LIN {X 0,Y 483.9,Z 922.544,A -85,B 0,C 180,E1 -6915.573,E2 -6915.573} C_VEL
LIN {X 0,Y 483.495,Z 935.94,A -85,B 0,C 180,E1 -6916.125,E2 -6916.125} C_VEL
LIN {X 0,Y 483.076,Z 947.548,A -85,B 0,C 180,E1 -6916.777,E2 -6916.777} C_VEL
LIN {X 0,Y 482.662,Z 958.984,A -85,B 0,C 180,E1 -6917.599,E2 -6917.599} C_VEL
LIN {X 0,Y 482.218,Z 969.588,A -85,B 0,C 180,E1 -6918.548,E2 -6918.548} C_VEL
LIN {X 0,Y 481.844,Z 978.283,A -85,B 0,C 180,E1 -6919.497,E2 -6919.497} C_VEL
LIN {X 0,Y 481.566,Z 986.33,A -85,B 0,C 180,E1 -6920.552,E2 -6920.552} C_VEL
LIN {X 0,Y 481.287,Z 994.208,A -85,B 0,C 180,E1 -6921.816,E2 -6921.816} C_VEL
LIN {X 0,Y 481.075,Z 1001.479,A -85,B 0,C 180,E1 -6923.29,E2 -6923.29} C_VEL
LIN {X 0,Y 481,Z 1006.335,A -85,B 0,C 180,E1 -6924.552,E2 -6924.552} C_VEL
LIN {X 0,Y 480.896,Z 1010.045,A -85,B 0,C 180,E1 -6925.811,E2 -6925.811} C_VEL
LIN {X 0,Y 480.923,Z 1011.97,A -85,B 0,C 180,E1 -6926.65,E2 -6926.65} C_VEL
LIN {X 0,Y 480.824,Z 1014.423,A -85,B 0,C 180,E1 -6928.326,E2 -6928.326} C_VEL
LIN {X 0,Y 480.773,Z 1015.041,A -85,B 0,C 180,E1 -6929.164,E2 -6929.164} C_VEL
LIN {X 0,Y 480.758,Z 1015.261,A -85,B 0,C 180,E1 -6930.001,E2 -6930.001} C_VEL
LIN {X 0,Y 480.773,Z 1015.039,A -85,B 0,C 180,E1 -6930.839,E2 -6930.839} C_VEL
LIN {X 0,Y 480.824,Z 1014.418,A -85,B 0,C 180,E1 -6931.677,E2 -6931.677} C_VEL
LIN {X 0,Y 480.924,Z 1011.961,A -85,B 0,C 180,E1 -6933.353,E2 -6933.353} C_VEL
LIN {X 0,Y 480.899,Z 1008.931,A -85,B 0,C 180,E1 -6934.612,E2 -6934.612} C_VEL
LIN {X 0,Y 481.047,Z 1004.858,A -85,B 0,C 180,E1 -6935.871,E2 -6935.871} C_VEL
LIN {X 0,Y 481.118,Z 998.567,A -85,B 0,C 180,E1 -6937.345,E2 -6937.345} C_VEL
LIN {X 0,Y 481.382,Z 991.735,A -85,B 0,C 180,E1 -6938.608,E2 -6938.608} C_VEL
LIN {X 0,Y 481.695,Z 983.271,A -85,B 0,C 180,E1 -6939.873,E2 -6939.873} C_VEL
LIN {X 0,Y 482.021,Z 974.606,A -85,B 0,C 180,E1 -6940.927,E2 -6940.927} C_VEL
LIN {X 0,Y 482.499,Z 963.942,A -85,B 0,C 180,E1 -6941.981,E2 -6941.981} C_VEL
LIN {X 0,Y 482.896,Z 952.218,A -85,B 0,C 180,E1 -6942.912,E2 -6942.912} C_VEL
LIN {X 0,Y 483.349,Z 939.937,A -85,B 0,C 180,E1 -6943.668,E2 -6943.668} C_VEL
LIN {X 0,Y 483.709,Z 927.469,A -85,B 0,C 180,E1 -6944.248,E2 -6944.248} C_VEL
LIN {X 0,Y 483.765,Z 919.717,A -85,B 0,C 180,E1 -6944.528,E2 -6944.528} C_VEL
LIN {X 0,Y 481.921,Z 906.606,A -85,B 0,C 180,E1 -6944.909,E2 -6944.909} C_VEL
LIN {X 0,Y 481.609,Z 903.06,A -85,B 0,C 180,E1 -6945.013,E2 -6945.013} C_VEL
LIN {X 0,Y 481.961,Z 889.747,A -85,B 0,C 180,E1 -6947.833,E2 -6947.833} C_VEL
LIN {X 0,Y 482.255,Z 874.313,A -85,B 0,C 180,E1 -6951.142,E2 -6951.142} C_VEL
LIN {X 0,Y 482.646,Z 860.861,A -85,B 0,C 180,E1 -6954.063,E2 -6954.063} C_VEL
LIN {X 0,Y 483.053,Z 846.87,A -85,B 0,C 180,E1 -6957.129,E2 -6957.129} C_VEL
LIN {X 0,Y 483.485,Z 831.351,A -85,B 0,C 180,E1 -6960.583,E2 -6960.583} C_VEL
LIN {X 0,Y 483.933,Z 818.655,A -85,B 0,C 180,E1 -6963.496,E2 -6963.496} C_VEL
LIN {X 0,Y 484.248,Z 807.022,A -85,B 0,C 180,E1 -6966.267,E2 -6966.267} C_VEL
LIN {X 0,Y 483.231,Z 800.666,A -85,B 0,C 180,E1 -6967.922,E2 -6967.922} C_VEL
LIN {X 0,Y 481.634,Z 792.492,A -85,B 0,C 180,E1 -6970.203,E2 -6970.203} C_VEL
LIN {X 0,Y 481.616,Z 792.493,A -85,B 0,C 180,E1 -6973.304,E2 -6973.304} C_VEL
LIN {X 0,Y 481.603,Z 792.499,A -85,B 0,C 180,E1 -6975.649,E2 -6975.649} C_VEL
LIN {X 0,Y 481.606,Z 792.492,A -85,B 0,C 180,E1 -6978.953,E2 -6978.953} C_VEL
LIN {X 0,Y 481.618,Z 792.494,A -85,B 0,C 180,E1 -6982,E2 -6982} C_VEL
LIN {X 0,Y 481.648,Z 792.488,A -85,B 0,C 180,E1 -6985.314,E2 -6985.314} C_VEL
LIN {X 0,Y 481.624,Z 792.492,A -85,B 0,C 180,E1 -6988.31,E2 -6988.31} C_VEL
LIN {X 0,Y 481.631,Z 792.488,A -85,B 0,C 180,E1 -6991.214,E2 -6991.214} C_VEL
LIN {X 0,Y 481.607,Z 792.496,A -85,B 0,C 180,E1 -6994.037,E2 -6994.037} C_VEL
LIN {X 0,Y 481.632,Z 792.488,A -85,B 0,C 180,E1 -6996.825,E2 -6996.825} C_VEL
LIN {X 0,Y 481.617,Z 792.491,A -85,B 0,C 180,E1 -6999.499,E2 -6999.499} C_VEL
LIN {X 0,Y 481.64,Z 792.493,A -85,B 0,C 180,E1 -7002.156,E2 -7002.156} C_VEL
LIN {X 0,Y 481.694,Z 792.486,A -85,B 0,C 180,E1 -7004.774,E2 -7004.774} C_VEL
LIN {X 0,Y 481.712,Z 792.618,A -85,B 0,C 180,E1 -7006.043,E2 -7006.043} C_VEL
LIN {X 0,Y 483.56,Z 799.412,A -85,B 0,C 180,E1 -7006.446,E2 -7006.446} C_VEL
LIN {X 0,Y 483.478,Z 810.921,A -85,B 0,C 180,E1 -7007.169,E2 -7007.169} C_VEL
LIN {X 0,Y 483.179,Z 820.671,A -85,B 0,C 180,E1 -7007.931,E2 -7007.931} C_VEL
LIN {X 0,Y 482.897,Z 828.589,A -85,B 0,C 180,E1 -7008.669,E2 -7008.669} C_VEL
LIN {X 0,Y 482.517,Z 837.913,A -85,B 0,C 180,E1 -7009.722,E2 -7009.722} C_VEL
LIN {X 0,Y 482.217,Z 845.434,A -85,B 0,C 180,E1 -7010.775,E2 -7010.775} C_VEL
LIN {X 0,Y 481.924,Z 851.738,A -85,B 0,C 180,E1 -7011.826,E2 -7011.826} C_VEL
LIN {X 0,Y 481.823,Z 856.164,A -85,B 0,C 180,E1 -7012.692,E2 -7012.692} C_VEL
LIN {X 0,Y 481.635,Z 862.067,A -85,B 0,C 180,E1 -7014.137,E2 -7014.137} C_VEL
LIN {X 0,Y 481.389,Z 864.819,A -85,B 0,C 180,E1 -7014.975,E2 -7014.975} C_VEL
LIN {X 0,Y 481.403,Z 866.963,A -85,B 0,C 180,E1 -7015.814,E2 -7015.814} C_VEL
LIN {X 0,Y 481.31,Z 870.195,A -85,B 0,C 180,E1 -7017.489,E2 -7017.489} C_VEL
LIN {X 0,Y 481.129,Z 871.712,A -85,B 0,C 180,E1 -7019.163,E2 -7019.163} C_VEL
LIN {X 0,Y 481.106,Z 871.896,A -85,B 0,C 180,E1 -7020,E2 -7020} C_VEL
LIN {X 0,Y 481.129,Z 871.66,A -85,B 0,C 180,E1 -7020.837,E2 -7020.837} C_VEL
LIN {X 0,Y 481.171,Z 869.996,A -85,B 0,C 180,E1 -7022.511,E2 -7022.511} C_VEL
LIN {X 0,Y 481.34,Z 866.697,A -85,B 0,C 180,E1 -7024.187,E2 -7024.187} C_VEL
LIN {X 0,Y 481.414,Z 863.086,A -85,B 0,C 180,E1 -7025.445,E2 -7025.445} C_VEL
LIN {X 0,Y 481.598,Z 858.349,A -85,B 0,C 180,E1 -7026.704,E2 -7026.704} C_VEL
LIN {X 0,Y 481.74,Z 853.505,A -85,B 0,C 180,E1 -7027.756,E2 -7027.756} C_VEL
LIN {X 0,Y 482.022,Z 846.333,A -85,B 0,C 180,E1 -7029.018,E2 -7029.018} C_VEL
LIN {X 0,Y 482.274,Z 838.919,A -85,B 0,C 180,E1 -7030.071,E2 -7030.071} C_VEL
LIN {X 0,Y 482.556,Z 831.974,A -85,B 0,C 180,E1 -7030.914,E2 -7030.914} C_VEL
LIN {X 0,Y 482.8,Z 823.76,A -85,B 0,C 180,E1 -7031.759,E2 -7031.759} C_VEL
LIN {X 0,Y 483.183,Z 813.877,A -85,B 0,C 180,E1 -7032.602,E2 -7032.602} C_VEL
LIN {X 0,Y 483.482,Z 803.895,A -85,B 0,C 180,E1 -7033.283,E2 -7033.283} C_VEL
LIN {X 0,Y 483.46,Z 799.397,A -85,B 0,C 180,E1 -7033.557,E2 -7033.557} C_VEL
LIN {X 0,Y 481.664,Z 792.488,A -85,B 0,C 180,E1 -7033.985,E2 -7033.985} C_VEL
LIN {X 0,Y 481.641,Z 792.489,A -85,B 0,C 180,E1 -7036.096,E2 -7036.096} C_VEL
LIN {X 0,Y 481.625,Z 792.487,A -85,B 0,C 180,E1 -7038.725,E2 -7038.725} C_VEL
LIN {X 0,Y 481.623,Z 792.489,A -85,B 0,C 180,E1 -7041.396,E2 -7041.396} C_VEL
LIN {X 0,Y 481.619,Z 792.49,A -85,B 0,C 180,E1 -7044.116,E2 -7044.116} C_VEL
LIN {X 0,Y 481.646,Z 792.482,A -85,B 0,C 180,E1 -7047.114,E2 -7047.114} C_VEL
LIN {X 0,Y 481.658,Z 792.489,A -85,B 0,C 180,E1 -7049.743,E2 -7049.743} C_VEL
LIN {X 0,Y 481.653,Z 792.479,A -85,B 0,C 180,E1 -7052.676,E2 -7052.676} C_VEL
LIN {X 0,Y 481.654,Z 792.483,A -85,B 0,C 180,E1 -7055.201,E2 -7055.201} C_VEL
LIN {X 0,Y 481.635,Z 792.49,A -85,B 0,C 180,E1 -7058.003,E2 -7058.003} C_VEL
LIN {X 0,Y 481.631,Z 792.485,A -85,B 0,C 180,E1 -7061.045,E2 -7061.045} C_VEL
LIN {X 0,Y 481.66,Z 792.485,A -85,B 0,C 180,E1 -7064.458,E2 -7064.458} C_VEL
LIN {X 0,Y 481.646,Z 792.489,A -85,B 0,C 180,E1 -7067.838,E2 -7067.838} C_VEL
LIN {X 0,Y 481.672,Z 792.481,A -85,B 0,C 180,E1 -7071.14,E2 -7071.14} C_VEL
LIN {X 0,Y 481.665,Z 792.483,A -85,B 0,C 180,E1 -7074.796,E2 -7074.796} C_VEL
LIN {X 0,Y 481.662,Z 792.485,A -85,B 0,C 180,E1 -7077.81,E2 -7077.81} C_VEL
LIN {X 0,Y 481.704,Z 792.474,A -85,B 0,C 180,E1 -7081.218,E2 -7081.218} C_VEL
LIN {X 0,Y 481.675,Z 792.482,A -85,B 0,C 180,E1 -7084.115,E2 -7084.115} C_VEL
LIN {X 0,Y 480.993,Z 792.565,A -85,B 0,C 180,E1 -7084.813,E2 -7084.813} C_VEL
LIN {X 0,Y 478.124,Z 792.922,A -85,B 0,C 180,E1 -7085.947,E2 -7085.947} C_VEL
LIN {X 0,Y 475.706,Z 793.227,A -85,B 0,C 180,E1 -7086.861,E2 -7086.861} C_VEL
LIN {X 0,Y 474.67,Z 793.354,A -85,B 0,C 180,E1 -7087.568,E2 -7087.568} C_VEL
LIN {X 0,Y 474.586,Z 793.366,A -85,B 0,C 180,E1 -7087.807,E2 -7087.807} C_VEL
LIN {X 0,Y 474.66,Z 793.361,A -85,B 0,C 180,E1 -7090.088,E2 -7090.088} C_VEL
LIN {X 0,Y 474.642,Z 793.365,A -85,B 0,C 180,E1 -7092.773,E2 -7092.773} C_VEL
LIN {X 0,Y 474.674,Z 793.357,A -85,B 0,C 180,E1 -7095.612,E2 -7095.612} C_VEL
LIN {X 0,Y 477.158,Z 802.152,A -85,B 0,C 180,E1 -7096.151,E2 -7096.151} C_VEL
LIN {X 0,Y 477.085,Z 812.643,A -85,B 0,C 180,E1 -7096.812,E2 -7096.812} C_VEL
LIN {X 0,Y 476.651,Z 823.432,A -85,B 0,C 180,E1 -7097.654,E2 -7097.654} C_VEL
LIN {X 0,Y 476.309,Z 832.277,A -85,B 0,C 180,E1 -7098.509,E2 -7098.509} C_VEL
LIN {X 0,Y 475.895,Z 841.339,A -85,B 0,C 180,E1 -7099.576,E2 -7099.576} C_VEL
LIN {X 0,Y 475.468,Z 850.111,A -85,B 0,C 180,E1 -7100.856,E2 -7100.856} C_VEL
LIN {X 0,Y 475.125,Z 857.159,A -85,B 0,C 180,E1 -7102.134,E2 -7102.134} C_VEL
LIN {X 0,Y 475.013,Z 861.893,A -85,B 0,C 180,E1 -7103.201,E2 -7103.201} C_VEL
LIN {X 0,Y 474.635,Z 866.527,A -85,B 0,C 180,E1 -7104.475,E2 -7104.475} C_VEL
LIN {X 0,Y 474.515,Z 870.043,A -85,B 0,C 180,E1 -7105.752,E2 -7105.752} C_VEL
LIN {X 0,Y 474.413,Z 871.866,A -85,B 0,C 180,E1 -7106.601,E2 -7106.601} C_VEL
LIN {X 0,Y 474.428,Z 873.229,A -85,B 0,C 180,E1 -7107.451,E2 -7107.451} C_VEL
LIN {X 0,Y 474.342,Z 874.81,A -85,B 0,C 180,E1 -7109.15,E2 -7109.15} C_VEL
LIN {X 0,Y 474.361,Z 875.038,A -85,B 0,C 180,E1 -7109.998,E2 -7109.998} C_VEL
LIN {X 0,Y 474.305,Z 874.304,A -85,B 0,C 180,E1 -7111.697,E2 -7111.697} C_VEL
LIN {X 0,Y 474.427,Z 873.352,A -85,B 0,C 180,E1 -7112.546,E2 -7112.546} C_VEL
LIN {X 0,Y 474.408,Z 872.043,A -85,B 0,C 180,E1 -7113.396,E2 -7113.396} C_VEL
LIN {X 0,Y 474.554,Z 869.241,A -85,B 0,C 180,E1 -7114.671,E2 -7114.671} C_VEL
LIN {X 0,Y 474.825,Z 865.428,A -85,B 0,C 180,E1 -7115.945,E2 -7115.945} C_VEL
LIN {X 0,Y 475.021,Z 860.484,A -85,B 0,C 180,E1 -7117.234,E2 -7117.234} C_VEL
LIN {X 0,Y 475.259,Z 854.356,A -85,B 0,C 180,E1 -7118.502,E2 -7118.502} C_VEL
LIN {X 0,Y 475.672,Z 846.595,A -85,B 0,C 180,E1 -7119.781,E2 -7119.781} C_VEL
LIN {X 0,Y 476.051,Z 838.675,A -85,B 0,C 180,E1 -7120.848,E2 -7120.848} C_VEL
LIN {X 0,Y 476.451,Z 828.997,A -85,B 0,C 180,E1 -7121.916,E2 -7121.916} C_VEL
LIN {X 0,Y 476.812,Z 819.458,A -85,B 0,C 180,E1 -7122.772,E2 -7122.772} C_VEL
LIN {X 0,Y 477.177,Z 808.266,A -85,B 0,C 180,E1 -7123.573,E2 -7123.573} C_VEL
LIN {X 0,Y 477.358,Z 803.815,A -85,B 0,C 180,E1 -7123.84,E2 -7123.84} C_VEL
LIN {X 0,Y 475.979,Z 797.969,A -85,B 0,C 180,E1 -7124.208,E2 -7124.208} C_VEL
LIN {X 0,Y 474.653,Z 793.36,A -85,B 0,C 180,E1 -7124.495,E2 -7124.495} C_VEL
LIN {X 0,Y 474.65,Z 793.361,A -85,B 0,C 180,E1 -7127.224,E2 -7127.224} C_VEL
LIN {X 0,Y 474.655,Z 793.362,A -85,B 0,C 180,E1 -7129.908,E2 -7129.908} C_VEL
LIN {X 0,Y 474.633,Z 793.361,A -85,B 0,C 180,E1 -7133.357,E2 -7133.357} C_VEL
LIN {X 0,Y 474.657,Z 793.358,A -85,B 0,C 180,E1 -7136.37,E2 -7136.37} C_VEL
LIN {X 0,Y 474.618,Z 793.361,A -85,B 0,C 180,E1 -7139.25,E2 -7139.25} C_VEL
LIN {X 0,Y 474.611,Z 793.365,A -85,B 0,C 180,E1 -7142.429,E2 -7142.429} C_VEL
LIN {X 0,Y 474.612,Z 793.362,A -85,B 0,C 180,E1 -7145.468,E2 -7145.468} C_VEL
LIN {X 0,Y 474.615,Z 793.366,A -85,B 0,C 180,E1 -7148.454,E2 -7148.454} C_VEL
LIN {X 0,Y 474.637,Z 793.358,A -85,B 0,C 180,E1 -7150.96,E2 -7150.96} C_VEL
LIN {X 0,Y 474.608,Z 793.367,A -85,B 0,C 180,E1 -7154.102,E2 -7154.102} C_VEL
LIN {X 0,Y 474.641,Z 793.355,A -85,B 0,C 180,E1 -7157.068,E2 -7157.068} C_VEL
LIN {X 0,Y 474.662,Z 793.361,A -85,B 0,C 180,E1 -7160.456,E2 -7160.456} C_VEL
LIN {X 0,Y 474.58,Z 793.364,A -85,B 0,C 180,E1 -7163.675,E2 -7163.675} C_VEL
LIN {X 0,Y 474.629,Z 793.365,A -85,B 0,C 180,E1 -7166.779,E2 -7166.779} C_VEL
LIN {X 0,Y 474.599,Z 793.359,A -85,B 0,C 180,E1 -7169.769,E2 -7169.769} C_VEL
LIN {X 0,Y 474.699,Z 793.357,A -85,B 0,C 180,E1 -7172.68,E2 -7172.68} C_VEL
LIN {X 0,Y 474.644,Z 793.357,A -85,B 0,C 180,E1 -7175.506,E2 -7175.506} C_VEL
LIN {X 0,Y 474.654,Z 793.359,A -85,B 0,C 180,E1 -7179.184,E2 -7179.184} C_VEL
LIN {X 0,Y 474.64,Z 793.357,A -85,B 0,C 180,E1 -7181.884,E2 -7181.884} C_VEL
LIN {X 0,Y 474.682,Z 793.35,A -85,B 0,C 180,E1 -7184.544,E2 -7184.544} C_VEL
LIN {X 0,Y 474.724,Z 793.347,A -85,B 0,C 180,E1 -7188.038,E2 -7188.038} C_VEL
LIN {X 0,Y 474.712,Z 793.354,A -85,B 0,C 180,E1 -7191.486,E2 -7191.486} C_VEL
LIN {X 0,Y 474.753,Z 793.345,A -85,B 0,C 180,E1 -7194.052,E2 -7194.052} C_VEL
LIN {X 0,Y 474.876,Z 793.334,A -85,B 0,C 180,E1 -7197.455,E2 -7197.455} C_VEL
LIN {X 0,Y 474.89,Z 793.33,A -85,B 0,C 180,E1 -7200,E2 -7200} C_VEL
LIN {X 0,Y 474.875,Z 793.329,A -85,B 0,C 180,E1 -7202.545,E2 -7202.545} C_VEL
LIN {X 0,Y 474.74,Z 793.349,A -85,B 0,C 180,E1 -7205.948,E2 -7205.948} C_VEL
LIN {X 0,Y 474.709,Z 793.348,A -85,B 0,C 180,E1 -7208.514,E2 -7208.514} C_VEL
LIN {X 0,Y 474.721,Z 793.35,A -85,B 0,C 180,E1 -7211.962,E2 -7211.962} C_VEL
LIN {X 0,Y 474.661,Z 793.362,A -85,B 0,C 180,E1 -7215.768,E2 -7215.768} C_VEL
LIN {X 0,Y 474.645,Z 793.357,A -85,B 0,C 180,E1 -7219.011,E2 -7219.011} C_VEL
LIN {X 0,Y 474.571,Z 793.371,A -85,B 0,C 180,E1 -7221.73,E2 -7221.73} C_VEL
LIN {X 0,Y 474.614,Z 793.363,A -85,B 0,C 180,E1 -7224.495,E2 -7224.495} C_VEL
LIN {X 0,Y 474.62,Z 793.359,A -85,B 0,C 180,E1 -7227.325,E2 -7227.325} C_VEL
LIN {X 0,Y 474.587,Z 793.37,A -85,B 0,C 180,E1 -7230.232,E2 -7230.232} C_VEL
LIN {X 0,Y 474.606,Z 793.362,A -85,B 0,C 180,E1 -7233.223,E2 -7233.223} C_VEL
LIN {X 0,Y 474.564,Z 793.375,A -85,B 0,C 180,E1 -7236.326,E2 -7236.326} C_VEL
LIN {X 0,Y 474.587,Z 793.366,A -85,B 0,C 180,E1 -7239.645,E2 -7239.645} C_VEL
LIN {X 0,Y 474.561,Z 793.373,A -85,B 0,C 180,E1 -7242.94,E2 -7242.94} C_VEL
LIN {X 0,Y 474.585,Z 793.368,A -85,B 0,C 180,E1 -7245.895,E2 -7245.895} C_VEL
LIN {X 0,Y 474.602,Z 793.368,A -85,B 0,C 180,E1 -7249.47,E2 -7249.47} C_VEL
LIN {X 0,Y 474.618,Z 793.527,A -85,B 0,C 180,E1 -7249.597,E2 -7249.597} C_VEL
LIN {X 0,Y 476.953,Z 805.247,A -85,B 0,C 180,E1 -7252.835,E2 -7252.835} C_VEL
LIN {X 0,Y 477.313,Z 810.127,A -85,B 0,C 180,E1 -7254.079,E2 -7254.079} C_VEL
LIN {X 0,Y 476.863,Z 822.093,A -85,B 0,C 180,E1 -7256.957,E2 -7256.957} C_VEL
LIN {X 0,Y 476.399,Z 834.791,A -85,B 0,C 180,E1 -7259.898,E2 -7259.898} C_VEL
LIN {X 0,Y 476.003,Z 848.539,A -85,B 0,C 180,E1 -7263.001,E2 -7263.001} C_VEL
LIN {X 0,Y 475.588,Z 862.135,A -85,B 0,C 180,E1 -7266.023,E2 -7266.023} C_VEL
LIN {X 0,Y 475.137,Z 877.652,A -85,B 0,C 180,E1 -7269.435,E2 -7269.435} C_VEL
LIN {X 0,Y 474.809,Z 891.946,A -85,B 0,C 180,E1 -7272.56,E2 -7272.56} C_VEL
LIN {X 0,Y 474.543,Z 902.182,A -85,B 0,C 180,E1 -7274.788,E2 -7274.788} C_VEL
LIN {X 0,Y 475.988,Z 914.958,A -85,B 0,C 180,E1 -7275.123,E2 -7275.123} C_VEL
LIN {X 0,Y 476.932,Z 923.027,A -85,B 0,C 180,E1 -7275.412,E2 -7275.412} C_VEL
LIN {X 0,Y 476.524,Z 935.928,A -85,B 0,C 180,E1 -7275.972,E2 -7275.972} C_VEL
LIN {X 0,Y 476.038,Z 948.259,A -85,B 0,C 180,E1 -7276.697,E2 -7276.697} C_VEL
LIN {X 0,Y 475.624,Z 959.269,A -85,B 0,C 180,E1 -7277.523,E2 -7277.523} C_VEL
LIN {X 0,Y 475.139,Z 969.601,A -85,B 0,C 180,E1 -7278.483,E2 -7278.483} C_VEL
LIN {X 0,Y 474.734,Z 978.948,A -85,B 0,C 180,E1 -7279.553,E2 -7279.553} C_VEL
LIN {X 0,Y 474.405,Z 988.081,A -85,B 0,C 180,E1 -7280.838,E2 -7280.838} C_VEL
LIN {X 0,Y 474.143,Z 995.45,A -85,B 0,C 180,E1 -7282.121,E2 -7282.121} C_VEL
LIN {X 0,Y 473.979,Z 1001.499,A -85,B 0,C 180,E1 -7283.442,E2 -7283.442} C_VEL
LIN {X 0,Y 473.893,Z 1006.643,A -85,B 0,C 180,E1 -7284.897,E2 -7284.897} C_VEL
LIN {X 0,Y 473.85,Z 1009.008,A -85,B 0,C 180,E1 -7285.749,E2 -7285.749} C_VEL
LIN {X 0,Y 473.881,Z 1010.935,A -85,B 0,C 180,E1 -7286.601,E2 -7286.601} C_VEL
LIN {X 0,Y 473.792,Z 1013.39,A -85,B 0,C 180,E1 -7288.302,E2 -7288.302} C_VEL
LIN {X 0,Y 473.747,Z 1014.009,A -85,B 0,C 180,E1 -7289.152,E2 -7289.152} C_VEL
LIN {X 0,Y 473.734,Z 1014.229,A -85,B 0,C 180,E1 -7290.002,E2 -7290.002} C_VEL
LIN {X 0,Y 473.747,Z 1014.007,A -85,B 0,C 180,E1 -7290.852,E2 -7290.852} C_VEL
LIN {X 0,Y 473.793,Z 1013.385,A -85,B 0,C 180,E1 -7291.702,E2 -7291.702} C_VEL
LIN {X 0,Y 473.882,Z 1010.925,A -85,B 0,C 180,E1 -7293.402,E2 -7293.402} C_VEL
LIN {X 0,Y 473.86,Z 1007.894,A -85,B 0,C 180,E1 -7294.68,E2 -7294.68} C_VEL
LIN {X 0,Y 473.989,Z 1003.816,A -85,B 0,C 180,E1 -7295.959,E2 -7295.959} C_VEL
LIN {X 0,Y 474.079,Z 997.525,A -85,B 0,C 180,E1 -7297.455,E2 -7297.455} C_VEL
LIN {X 0,Y 474.333,Z 990.688,A -85,B 0,C 180,E1 -7298.737,E2 -7298.737} C_VEL
LIN {X 0,Y 474.628,Z 982.217,A -85,B 0,C 180,E1 -7300.021,E2 -7300.021} C_VEL
LIN {X 0,Y 475.01,Z 973.557,A -85,B 0,C 180,E1 -7301.091,E2 -7301.091} C_VEL
LIN {X 0,Y 475.52,Z 962.895,A -85,B 0,C 180,E1 -7302.159,E2 -7302.159} C_VEL
LIN {X 0,Y 475.901,Z 951.335,A -85,B 0,C 180,E1 -7303.092,E2 -7303.092} C_VEL
LIN {X 0,Y 476.385,Z 938.884,A -85,B 0,C 180,E1 -7303.872,E2 -7303.872} C_VEL
LIN {X 0,Y 476.79,Z 926.421,A -85,B 0,C 180,E1 -7304.459,E2 -7304.459} C_VEL
LIN {X 0,Y 476.773,Z 920.23,A -85,B 0,C 180,E1 -7304.691,E2 -7304.691} C_VEL
LIN {X 0,Y 475.08,Z 907.695,A -85,B 0,C 180,E1 -7305.087,E2 -7305.087} C_VEL
LIN {X 0,Y 474.548,Z 902.188,A -85,B 0,C 180,E1 -7305.215,E2 -7305.215} C_VEL
LIN {X 0,Y 474.929,Z 887.43,A -85,B 0,C 180,E1 -7308.416,E2 -7308.416} C_VEL
LIN {X 0,Y 475.218,Z 874.257,A -85,B 0,C 180,E1 -7311.297,E2 -7311.297} C_VEL
LIN {X 0,Y 475.622,Z 861.091,A -85,B 0,C 180,E1 -7314.209,E2 -7314.209} C_VEL
LIN {X 0,Y 476.027,Z 847.465,A -85,B 0,C 180,E1 -7317.239,E2 -7317.239} C_VEL
LIN {X 0,Y 476.482,Z 832.656,A -85,B 0,C 180,E1 -7320.59,E2 -7320.59} C_VEL
LIN {X 0,Y 476.977,Z 819.963,A -85,B 0,C 180,E1 -7323.543,E2 -7323.543} C_VEL
LIN {X 0,Y 477.336,Z 808.396,A -85,B 0,C 180,E1 -7326.344,E2 -7326.344} C_VEL
LIN {X 0,Y 476.279,Z 802.037,A -85,B 0,C 180,E1 -7328.03,E2 -7328.03} C_VEL
LIN {X 0,Y 474.597,Z 793.369,A -85,B 0,C 180,E1 -7330.471,E2 -7330.471} C_VEL
LIN {X 0,Y 474.562,Z 793.371,A -85,B 0,C 180,E1 -7333.476,E2 -7333.476} C_VEL
LIN {X 0,Y 474.546,Z 793.371,A -85,B 0,C 180,E1 -7336.527,E2 -7336.527} C_VEL
LIN {X 0,Y 474.571,Z 793.373,A -85,B 0,C 180,E1 -7339.337,E2 -7339.337} C_VEL
LIN {X 0,Y 474.583,Z 793.37,A -85,B 0,C 180,E1 -7341.71,E2 -7341.71} C_VEL
LIN {X 0,Y 474.571,Z 793.367,A -85,B 0,C 180,E1 -7344.721,E2 -7344.721} C_VEL
LIN {X 0,Y 474.614,Z 793.366,A -85,B 0,C 180,E1 -7347.786,E2 -7347.786} C_VEL
LIN {X 0,Y 474.577,Z 793.367,A -85,B 0,C 180,E1 -7350.897,E2 -7350.897} C_VEL
LIN {X 0,Y 474.559,Z 793.372,A -85,B 0,C 180,E1 -7353.622,E2 -7353.622} C_VEL
LIN {X 0,Y 474.599,Z 793.366,A -85,B 0,C 180,E1 -7356.654,E2 -7356.654} C_VEL
LIN {X 0,Y 474.618,Z 793.363,A -85,B 0,C 180,E1 -7359.183,E2 -7359.183} C_VEL
LIN {X 0,Y 474.594,Z 793.369,A -85,B 0,C 180,E1 -7361.882,E2 -7361.882} C_VEL
LIN {X 0,Y 474.654,Z 793.364,A -85,B 0,C 180,E1 -7364.543,E2 -7364.543} C_VEL
LIN {X 0,Y 474.638,Z 793.364,A -85,B 0,C 180,E1 -7365.804,E2 -7365.804} C_VEL
LIN {X 0,Y 476.853,Z 802.263,A -85,B 0,C 180,E1 -7366.36,E2 -7366.36} C_VEL
LIN {X 0,Y 476.602,Z 813.02,A -85,B 0,C 180,E1 -7367.063,E2 -7367.063} C_VEL
LIN {X 0,Y 476.258,Z 822.874,A -85,B 0,C 180,E1 -7367.861,E2 -7367.861} C_VEL
LIN {X 0,Y 476.029,Z 829.646,A -85,B 0,C 180,E1 -7368.503,E2 -7368.503} C_VEL
LIN {X 0,Y 475.628,Z 838.964,A -85,B 0,C 180,E1 -7369.571,E2 -7369.571} C_VEL
LIN {X 0,Y 475.289,Z 846.504,A -85,B 0,C 180,E1 -7370.639,E2 -7370.639} C_VEL
LIN {X 0,Y 474.979,Z 852.816,A -85,B 0,C 180,E1 -7371.705,E2 -7371.705} C_VEL
LIN {X 0,Y 474.865,Z 857.199,A -85,B 0,C 180,E1 -7372.573,E2 -7372.573} C_VEL
LIN {X 0,Y 474.662,Z 863.15,A -85,B 0,C 180,E1 -7374.051,E2 -7374.051} C_VEL
LIN {X 0,Y 474.402,Z 865.908,A -85,B 0,C 180,E1 -7374.9,E2 -7374.9} C_VEL
LIN {X 0,Y 474.404,Z 868.049,A -85,B 0,C 180,E1 -7375.752,E2 -7375.752} C_VEL
LIN {X 0,Y 474.31,Z 871.277,A -85,B 0,C 180,E1 -7377.452,E2 -7377.452} C_VEL
LIN {X 0,Y 474.115,Z 872.783,A -85,B 0,C 180,E1 -7379.151,E2 -7379.151} C_VEL
LIN {X 0,Y 474.09,Z 872.959,A -85,B 0,C 180,E1 -7380,E2 -7380} C_VEL
LIN {X 0,Y 474.115,Z 872.714,A -85,B 0,C 180,E1 -7380.849,E2 -7380.849} C_VEL
LIN {X 0,Y 474.154,Z 871.025,A -85,B 0,C 180,E1 -7382.549,E2 -7382.549} C_VEL
LIN {X 0,Y 474.33,Z 867.692,A -85,B 0,C 180,E1 -7384.249,E2 -7384.249} C_VEL
LIN {X 0,Y 474.421,Z 864.051,A -85,B 0,C 180,E1 -7385.526,E2 -7385.526} C_VEL
LIN {X 0,Y 474.617,Z 859.281,A -85,B 0,C 180,E1 -7386.803,E2 -7386.803} C_VEL
LIN {X 0,Y 474.776,Z 854.405,A -85,B 0,C 180,E1 -7387.87,E2 -7387.87} C_VEL
LIN {X 0,Y 475.077,Z 847.198,A -85,B 0,C 180,E1 -7389.151,E2 -7389.151} C_VEL
LIN {X 0,Y 475.34,Z 839.741,A -85,B 0,C 180,E1 -7390.22,E2 -7390.22} C_VEL
LIN {X 0,Y 475.641,Z 832.756,A -85,B 0,C 180,E1 -7391.075,E2 -7391.075} C_VEL
LIN {X 0,Y 475.896,Z 824.497,A -85,B 0,C 180,E1 -7391.932,E2 -7391.932} C_VEL
LIN {X 0,Y 476.351,Z 813.356,A -85,B 0,C 180,E1 -7392.883,E2 -7392.883} C_VEL
LIN {X 0,Y 476.655,Z 803.186,A -85,B 0,C 180,E1 -7393.559,E2 -7393.559} C_VEL
LIN {X 0,Y 476.406,Z 800.049,A -85,B 0,C 180,E1 -7393.761,E2 -7393.761} C_VEL
LIN {X 0,Y 474.639,Z 793.362,A -85,B 0,C 180,E1 -7394.196,E2 -7394.196} C_VEL
LIN {X 0,Y 474.592,Z 793.365,A -85,B 0,C 180,E1 -7396.342,E2 -7396.342} C_VEL
LIN {X 0,Y 474.582,Z 793.365,A -85,B 0,C 180,E1 -7399.014,E2 -7399.014} C_VEL
LIN {X 0,Y 474.572,Z 793.369,A -85,B 0,C 180,E1 -7401.73,E2 -7401.73} C_VEL
LIN {X 0,Y 474.586,Z 793.364,A -85,B 0,C 180,E1 -7404.497,E2 -7404.497} C_VEL
LIN {X 0,Y 474.598,Z 793.361,A -85,B 0,C 180,E1 -7407.327,E2 -7407.327} C_VEL
LIN {X 0,Y 474.589,Z 793.365,A -85,B 0,C 180,E1 -7410.231,E2 -7410.231} C_VEL
LIN {X 0,Y 474.618,Z 793.356,A -85,B 0,C 180,E1 -7413.222,E2 -7413.222} C_VEL
LIN {X 0,Y 474.575,Z 793.366,A -85,B 0,C 180,E1 -7416.325,E2 -7416.325} C_VEL
LIN {X 0,Y 474.606,Z 793.364,A -85,B 0,C 180,E1 -7419.643,E2 -7419.643} C_VEL
LIN {X 0,Y 474.58,Z 793.363,A -85,B 0,C 180,E1 -7422.938,E2 -7422.938} C_VEL
LIN {X 0,Y 474.609,Z 793.367,A -85,B 0,C 180,E1 -7425.894,E2 -7425.894} C_VEL
LIN {X 0,Y 474.613,Z 793.36,A -85,B 0,C 180,E1 -7429.043,E2 -7429.043} C_VEL
LIN {X 0,Y 474.612,Z 793.364,A -85,B 0,C 180,E1 -7431.704,E2 -7431.704} C_VEL
LIN {X 0,Y 474.627,Z 793.361,A -85,B 0,C 180,E1 -7434.725,E2 -7434.725} C_VEL
LIN {X 0,Y 474.641,Z 793.359,A -85,B 0,C 180,E1 -7437.787,E2 -7437.787} C_VEL
LIN {X 0,Y 474.628,Z 793.357,A -85,B 0,C 180,E1 -7440.884,E2 -7440.884} C_VEL
LIN {X 0,Y 474.633,Z 793.356,A -85,B 0,C 180,E1 -7443.626,E2 -7443.626} C_VEL
LIN {X 0,Y 474.64,Z 793.363,A -85,B 0,C 180,E1 -7446.641,E2 -7446.641} C_VEL
LIN {X 0,Y 474.586,Z 793.366,A -85,B 0,C 180,E1 -7447.807,E2 -7447.807} C_VEL
LIN {X 0,Y 473.921,Z 793.455,A -85,B 0,C 180,E1 -7448.515,E2 -7448.515} C_VEL
LIN {X 0,Y 471.082,Z 793.807,A -85,B 0,C 180,E1 -7449.666,E2 -7449.666} C_VEL
LIN {X 0,Y 468.698,Z 794.107,A -85,B 0,C 180,E1 -7450.594,E2 -7450.594} C_VEL
LIN {X 0,Y 467.697,Z 794.227,A -85,B 0,C 180,E1 -7451.311,E2 -7451.311} C_VEL
LIN {X 0,Y 467.627,Z 794.235,A -85,B 0,C 180,E1 -7451.553,E2 -7451.553} C_VEL
LIN {X 0,Y 467.645,Z 794.235,A -85,B 0,C 180,E1 -7454.304,E2 -7454.304} C_VEL
LIN {X 0,Y 467.649,Z 794.397,A -85,B 0,C 180,E1 -7455.391,E2 -7455.391} C_VEL
LIN {X 0,Y 470.186,Z 803.216,A -85,B 0,C 180,E1 -7455.941,E2 -7455.941} C_VEL
LIN {X 0,Y 470.431,Z 806.901,A -85,B 0,C 180,E1 -7456.169,E2 -7456.169} C_VEL
LIN {X 0,Y 470.131,Z 817.479,A -85,B 0,C 180,E1 -7456.898,E2 -7456.898} C_VEL
LIN {X 0,Y 469.646,Z 827.956,A -85,B 0,C 180,E1 -7457.796,E2 -7457.796} C_VEL
LIN {X 0,Y 469.244,Z 837.16,A -85,B 0,C 180,E1 -7458.771,E2 -7458.771} C_VEL
LIN {X 0,Y 468.836,Z 845.541,A -85,B 0,C 180,E1 -7459.854,E2 -7459.854} C_VEL
LIN {X 0,Y 468.367,Z 853.668,A -85,B 0,C 180,E1 -7461.151,E2 -7461.151} C_VEL
LIN {X 0,Y 468.089,Z 859.443,A -85,B 0,C 180,E1 -7462.284,E2 -7462.284} C_VEL
LIN {X 0,Y 467.961,Z 864.59,A -85,B 0,C 180,E1 -7463.531,E2 -7463.531} C_VEL
LIN {X 0,Y 467.559,Z 868.851,A -85,B 0,C 180,E1 -7464.824,E2 -7464.824} C_VEL
LIN {X 0,Y 467.509,Z 871.075,A -85,B 0,C 180,E1 -7465.688,E2 -7465.688} C_VEL
LIN {X 0,Y 467.402,Z 872.898,A -85,B 0,C 180,E1 -7466.55,E2 -7466.55} C_VEL
LIN {X 0,Y 467.418,Z 874.26,A -85,B 0,C 180,E1 -7467.413,E2 -7467.413} C_VEL
LIN {X 0,Y 467.333,Z 875.839,A -85,B 0,C 180,E1 -7469.137,E2 -7469.137} C_VEL
LIN {X 0,Y 467.347,Z 876.068,A -85,B 0,C 180,E1 -7469.998,E2 -7469.998} C_VEL
LIN {X 0,Y 467.289,Z 875.334,A -85,B 0,C 180,E1 -7471.722,E2 -7471.722} C_VEL
LIN {X 0,Y 467.416,Z 874.381,A -85,B 0,C 180,E1 -7472.584,E2 -7472.584} C_VEL
LIN {X 0,Y 467.396,Z 873.073,A -85,B 0,C 180,E1 -7473.447,E2 -7473.447} C_VEL
LIN {X 0,Y 467.551,Z 870.272,A -85,B 0,C 180,E1 -7474.741,E2 -7474.741} C_VEL
LIN {X 0,Y 467.85,Z 866.456,A -85,B 0,C 180,E1 -7476.034,E2 -7476.034} C_VEL
LIN {X 0,Y 468.063,Z 861.459,A -85,B 0,C 180,E1 -7477.355,E2 -7477.355} C_VEL
LIN {X 0,Y 468.319,Z 855.384,A -85,B 0,C 180,E1 -7478.629,E2 -7478.629} C_VEL
LIN {X 0,Y 468.754,Z 847.622,A -85,B 0,C 180,E1 -7479.927,E2 -7479.927} C_VEL
LIN {X 0,Y 469.158,Z 839.702,A -85,B 0,C 180,E1 -7481.009,E2 -7481.009} C_VEL
LIN {X 0,Y 469.58,Z 830.024,A -85,B 0,C 180,E1 -7482.093,E2 -7482.093} C_VEL
LIN {X 0,Y 469.966,Z 820.484,A -85,B 0,C 180,E1 -7482.961,E2 -7482.961} C_VEL
LIN {X 0,Y 470.35,Z 809.276,A -85,B 0,C 180,E1 -7483.775,E2 -7483.775} C_VEL
LIN {X 0,Y 470.511,Z 804.842,A -85,B 0,C 180,E1 -7484.046,E2 -7484.046} C_VEL
LIN {X 0,Y 467.626,Z 794.235,A -85,B 0,C 180,E1 -7484.718,E2 -7484.718} C_VEL
LIN {X 0,Y 467.608,Z 794.241,A -85,B 0,C 180,E1 -7487.491,E2 -7487.491} C_VEL
LIN {X 0,Y 467.622,Z 794.234,A -85,B 0,C 180,E1 -7490.221,E2 -7490.221} C_VEL
LIN {X 0,Y 467.571,Z 794.245,A -85,B 0,C 180,E1 -7493.941,E2 -7493.941} C_VEL
LIN {X 0,Y 467.612,Z 794.233,A -85,B 0,C 180,E1 -7496.798,E2 -7496.798} C_VEL
LIN {X 0,Y 467.551,Z 794.246,A -85,B 0,C 180,E1 -7499.736,E2 -7499.736} C_VEL
LIN {X 0,Y 467.578,Z 794.238,A -85,B 0,C 180,E1 -7502.756,E2 -7502.756} C_VEL
LIN {X 0,Y 467.549,Z 794.247,A -85,B 0,C 180,E1 -7505.888,E2 -7505.888} C_VEL
LIN {X 0,Y 467.591,Z 794.236,A -85,B 0,C 180,E1 -7509.141,E2 -7509.141} C_VEL
LIN {X 0,Y 467.609,Z 794.238,A -85,B 0,C 180,E1 -7512.57,E2 -7512.57} C_VEL
LIN {X 0,Y 467.564,Z 794.245,A -85,B 0,C 180,E1 -7516.175,E2 -7516.175} C_VEL
LIN {X 0,Y 467.578,Z 794.242,A -85,B 0,C 180,E1 -7518.72,E2 -7518.72} C_VEL
LIN {X 0,Y 467.566,Z 794.236,A -85,B 0,C 180,E1 -7521.405,E2 -7521.405} C_VEL
LIN {X 0,Y 467.55,Z 794.244,A -85,B 0,C 180,E1 -7524.259,E2 -7524.259} C_VEL
LIN {X 0,Y 467.568,Z 794.239,A -85,B 0,C 180,E1 -7527.319,E2 -7527.319} C_VEL
LIN {X 0,Y 467.563,Z 794.243,A -85,B 0,C 180,E1 -7530.664,E2 -7530.664} C_VEL
LIN {X 0,Y 467.612,Z 794.234,A -85,B 0,C 180,E1 -7533.199,E2 -7533.199} C_VEL
LIN {X 0,Y 467.577,Z 794.239,A -85,B 0,C 180,E1 -7536.467,E2 -7536.467} C_VEL
LIN {X 0,Y 467.606,Z 794.232,A -85,B 0,C 180,E1 -7539.776,E2 -7539.776} C_VEL
LIN {X 0,Y 467.592,Z 794.237,A -85,B 0,C 180,E1 -7542.506,E2 -7542.506} C_VEL
LIN {X 0,Y 467.589,Z 794.239,A -85,B 0,C 180,E1 -7545.196,E2 -7545.196} C_VEL
LIN {X 0,Y 467.667,Z 794.227,A -85,B 0,C 180,E1 -7547.855,E2 -7547.855} C_VEL
LIN {X 0,Y 467.666,Z 794.231,A -85,B 0,C 180,E1 -7551.357,E2 -7551.357} C_VEL
LIN {X 0,Y 467.718,Z 794.222,A -85,B 0,C 180,E1 -7553.962,E2 -7553.962} C_VEL
LIN {X 0,Y 467.841,Z 794.21,A -85,B 0,C 180,E1 -7557.417,E2 -7557.417} C_VEL
LIN {X 0,Y 467.862,Z 794.205,A -85,B 0,C 180,E1 -7560,E2 -7560} C_VEL
LIN {X 0,Y 467.841,Z 794.206,A -85,B 0,C 180,E1 -7562.583,E2 -7562.583} C_VEL
LIN {X 0,Y 467.702,Z 794.224,A -85,B 0,C 180,E1 -7566.038,E2 -7566.038} C_VEL
LIN {X 0,Y 467.663,Z 794.226,A -85,B 0,C 180,E1 -7568.643,E2 -7568.643} C_VEL
LIN {X 0,Y 467.665,Z 794.227,A -85,B 0,C 180,E1 -7572.145,E2 -7572.145} C_VEL
LIN {X 0,Y 467.631,Z 794.238,A -85,B 0,C 180,E1 -7575.885,E2 -7575.885} C_VEL
LIN {X 0,Y 467.604,Z 794.236,A -85,B 0,C 180,E1 -7579.309,E2 -7579.309} C_VEL
LIN {X 0,Y 467.517,Z 794.253,A -85,B 0,C 180,E1 -7582.075,E2 -7582.075} C_VEL
LIN {X 0,Y 467.553,Z 794.24,A -85,B 0,C 180,E1 -7584.89,E2 -7584.89} C_VEL
LIN {X 0,Y 467.563,Z 794.241,A -85,B 0,C 180,E1 -7587.773,E2 -7587.773} C_VEL
LIN {X 0,Y 467.552,Z 794.241,A -85,B 0,C 180,E1 -7591.046,E2 -7591.046} C_VEL
LIN {X 0,Y 467.561,Z 794.247,A -85,B 0,C 180,E1 -7594.241,E2 -7594.241} C_VEL
LIN {X 0,Y 467.507,Z 794.248,A -85,B 0,C 180,E1 -7597.183,E2 -7597.183} C_VEL
LIN {X 0,Y 467.543,Z 794.247,A -85,B 0,C 180,E1 -7600.268,E2 -7600.268} C_VEL
LIN {X 0,Y 467.533,Z 794.246,A -85,B 0,C 180,E1 -7603.747,E2 -7603.747} C_VEL
LIN {X 0,Y 467.519,Z 794.249,A -85,B 0,C 180,E1 -7606.254,E2 -7606.254} C_VEL
LIN {X 0,Y 467.562,Z 794.443,A -85,B 0,C 180,E1 -7609.312,E2 -7609.312} C_VEL
LIN {X 0,Y 469.794,Z 805.571,A -85,B 0,C 180,E1 -7612.454,E2 -7612.454} C_VEL
LIN {X 0,Y 470.425,Z 810.591,A -85,B 0,C 180,E1 -7613.779,E2 -7613.779} C_VEL
LIN {X 0,Y 469.982,Z 821.3,A -85,B 0,C 180,E1 -7616.409,E2 -7616.409} C_VEL
LIN {X 0,Y 469.509,Z 833.967,A -85,B 0,C 180,E1 -7619.409,E2 -7619.409} C_VEL
LIN {X 0,Y 468.999,Z 848.742,A -85,B 0,C 180,E1 -7622.806,E2 -7622.806} C_VEL
LIN {X 0,Y 468.555,Z 862.336,A -85,B 0,C 180,E1 -7625.877,E2 -7625.877} C_VEL
LIN {X 0,Y 468.074,Z 877.784,A -85,B 0,C 180,E1 -7629.34,E2 -7629.34} C_VEL
LIN {X 0,Y 467.718,Z 892.051,A -85,B 0,C 180,E1 -7632.513,E2 -7632.513} C_VEL
LIN {X 0,Y 467.481,Z 901.107,A -85,B 0,C 180,E1 -7634.553,E2 -7634.553} C_VEL
LIN {X 0,Y 468.841,Z 913.872,A -85,B 0,C 180,E1 -7634.891,E2 -7634.891} C_VEL
LIN {X 0,Y 470.012,Z 922.747,A -85,B 0,C 180,E1 -7635.22,E2 -7635.22} C_VEL
LIN {X 0,Y 469.598,Z 934.879,A -85,B 0,C 180,E1 -7635.761,E2 -7635.761} C_VEL
LIN {X 0,Y 469.073,Z 946.724,A -85,B 0,C 180,E1 -7636.463,E2 -7636.463} C_VEL
LIN {X 0,Y 468.574,Z 958.512,A -85,B 0,C 180,E1 -7637.358,E2 -7637.358} C_VEL
LIN {X 0,Y 468.115,Z 968.548,A -85,B 0,C 180,E1 -7638.308,E2 -7638.308} C_VEL
LIN {X 0,Y 467.702,Z 977.898,A -85,B 0,C 180,E1 -7639.394,E2 -7639.394} C_VEL
LIN {X 0,Y 467.345,Z 987.031,A -85,B 0,C 180,E1 -7640.698,E2 -7640.698} C_VEL
LIN {X 0,Y 467.081,Z 994.403,A -85,B 0,C 180,E1 -7642.001,E2 -7642.001} C_VEL
LIN {X 0,Y 466.933,Z 1000.722,A -85,B 0,C 180,E1 -7643.412,E2 -7643.412} C_VEL
LIN {X 0,Y 466.842,Z 1005.603,A -85,B 0,C 180,E1 -7644.819,E2 -7644.819} C_VEL
LIN {X 0,Y 466.806,Z 1007.971,A -85,B 0,C 180,E1 -7645.684,E2 -7645.684} C_VEL
LIN {X 0,Y 466.84,Z 1009.899,A -85,B 0,C 180,E1 -7646.549,E2 -7646.549} C_VEL
LIN {X 0,Y 466.768,Z 1011.331,A -85,B 0,C 180,E1 -7647.413,E2 -7647.413} C_VEL
LIN {X 0,Y 466.761,Z 1012.357,A -85,B 0,C 180,E1 -7648.276,E2 -7648.276} C_VEL
LIN {X 0,Y 466.721,Z 1012.978,A -85,B 0,C 180,E1 -7649.139,E2 -7649.139} C_VEL
LIN {X 0,Y 466.71,Z 1013.198,A -85,B 0,C 180,E1 -7650.002,E2 -7650.002} C_VEL
LIN {X 0,Y 466.721,Z 1012.976,A -85,B 0,C 180,E1 -7650.864,E2 -7650.864} C_VEL
LIN {X 0,Y 466.761,Z 1012.353,A -85,B 0,C 180,E1 -7651.727,E2 -7651.727} C_VEL
LIN {X 0,Y 466.769,Z 1011.324,A -85,B 0,C 180,E1 -7652.59,E2 -7652.59} C_VEL
LIN {X 0,Y 466.841,Z 1009.89,A -85,B 0,C 180,E1 -7653.454,E2 -7653.454} C_VEL
LIN {X 0,Y 466.825,Z 1006.858,A -85,B 0,C 180,E1 -7654.751,E2 -7654.751} C_VEL
LIN {X 0,Y 466.931,Z 1002.774,A -85,B 0,C 180,E1 -7656.049,E2 -7656.049} C_VEL
LIN {X 0,Y 467.01,Z 996.479,A -85,B 0,C 180,E1 -7657.568,E2 -7657.568} C_VEL
LIN {X 0,Y 467.248,Z 989.635,A -85,B 0,C 180,E1 -7658.87,E2 -7658.87} C_VEL
LIN {X 0,Y 467.576,Z 981.166,A -85,B 0,C 180,E1 -7660.174,E2 -7660.174} C_VEL
LIN {X 0,Y 468.013,Z 972.511,A -85,B 0,C 180,E1 -7661.259,E2 -7661.259} C_VEL
LIN {X 0,Y 468.465,Z 963.171,A -85,B 0,C 180,E1 -7662.223,E2 -7662.223} C_VEL
LIN {X 0,Y 468.894,Z 951.296,A -85,B 0,C 180,E1 -7663.215,E2 -7663.215} C_VEL
LIN {X 0,Y 469.36,Z 939.784,A -85,B 0,C 180,E1 -7663.973,E2 -7663.973} C_VEL
LIN {X 0,Y 469.788,Z 927.994,A -85,B 0,C 180,E1 -7664.568,E2 -7664.568} C_VEL
LIN {X 0,Y 469.85,Z 921.105,A -85,B 0,C 180,E1 -7664.843,E2 -7664.843} C_VEL
LIN {X 0,Y 468.235,Z 908.954,A -85,B 0,C 180,E1 -7665.258,E2 -7665.258} C_VEL
LIN {X 0,Y 467.487,Z 901.171,A -85,B 0,C 180,E1 -7665.45,E2 -7665.45} C_VEL
LIN {X 0,Y 467.864,Z 886.891,A -85,B 0,C 180,E1 -7668.625,E2 -7668.625} C_VEL
LIN {X 0,Y 468.178,Z 873.156,A -85,B 0,C 180,E1 -7671.697,E2 -7671.697} C_VEL
LIN {X 0,Y 468.614,Z 860.24,A -85,B 0,C 180,E1 -7674.595,E2 -7674.595} C_VEL
LIN {X 0,Y 469.012,Z 847.666,A -85,B 0,C 180,E1 -7677.439,E2 -7677.439} C_VEL
LIN {X 0,Y 469.575,Z 832.096,A -85,B 0,C 180,E1 -7681.029,E2 -7681.029} C_VEL
LIN {X 0,Y 470.131,Z 818.13,A -85,B 0,C 180,E1 -7684.357,E2 -7684.357} C_VEL
LIN {X 0,Y 470.419,Z 810.573,A -85,B 0,C 180,E1 -7686.22,E2 -7686.22} C_VEL
LIN {X 0,Y 469.545,Z 804.421,A -85,B 0,C 180,E1 -7687.857,E2 -7687.857} C_VEL
LIN {X 0,Y 467.545,Z 794.249,A -85,B 0,C 180,E1 -7690.765,E2 -7690.765} C_VEL
LIN {X 0,Y 467.522,Z 794.248,A -85,B 0,C 180,E1 -7693.817,E2 -7693.817} C_VEL
LIN {X 0,Y 467.498,Z 794.25,A -85,B 0,C 180,E1 -7696.249,E2 -7696.249} C_VEL
LIN {X 0,Y 467.553,Z 794.242,A -85,B 0,C 180,E1 -7698.728,E2 -7698.728} C_VEL
LIN {X 0,Y 467.533,Z 794.249,A -85,B 0,C 180,E1 -7701.952,E2 -7701.952} C_VEL
LIN {X 0,Y 467.521,Z 794.247,A -85,B 0,C 180,E1 -7705.164,E2 -7705.164} C_VEL
LIN {X 0,Y 467.547,Z 794.247,A -85,B 0,C 180,E1 -7708.257,E2 -7708.257} C_VEL
LIN {X 0,Y 467.523,Z 794.246,A -85,B 0,C 180,E1 -7711.247,E2 -7711.247} C_VEL
LIN {X 0,Y 467.561,Z 794.245,A -85,B 0,C 180,E1 -7714.407,E2 -7714.407} C_VEL
LIN {X 0,Y 467.548,Z 794.242,A -85,B 0,C 180,E1 -7716.994,E2 -7716.994} C_VEL
LIN {X 0,Y 467.533,Z 794.248,A -85,B 0,C 180,E1 -7719.773,E2 -7719.773} C_VEL
LIN {X 0,Y 467.545,Z 794.249,A -85,B 0,C 180,E1 -7722.504,E2 -7722.504} C_VEL
LIN {X 0,Y 467.584,Z 794.242,A -85,B 0,C 180,E1 -7725.557,E2 -7725.557} C_VEL
LIN {X 0,Y 470.034,Z 803.398,A -85,B 0,C 180,E1 -7726.159,E2 -7726.159} C_VEL
LIN {X 0,Y 469.773,Z 814.134,A -85,B 0,C 180,E1 -7726.872,E2 -7726.872} C_VEL
LIN {X 0,Y 469.401,Z 823.985,A -85,B 0,C 180,E1 -7727.681,E2 -7727.681} C_VEL
LIN {X 0,Y 469.086,Z 832.678,A -85,B 0,C 180,E1 -7728.55,E2 -7728.55} C_VEL
LIN {X 0,Y 468.669,Z 841.745,A -85,B 0,C 180,E1 -7729.633,E2 -7729.633} C_VEL
LIN {X 0,Y 468.325,Z 848.949,A -85,B 0,C 180,E1 -7730.716,E2 -7730.716} C_VEL
LIN {X 0,Y 468.042,Z 853.923,A -85,B 0,C 180,E1 -7731.581,E2 -7731.581} C_VEL
LIN {X 0,Y 467.954,Z 858.075,A -85,B 0,C 180,E1 -7732.409,E2 -7732.409} C_VEL
LIN {X 0,Y 467.688,Z 864.253,A -85,B 0,C 180,E1 -7733.962,E2 -7733.962} C_VEL
LIN {X 0,Y 467.417,Z 867.01,A -85,B 0,C 180,E1 -7734.824,E2 -7734.824} C_VEL
LIN {X 0,Y 467.285,Z 870.931,A -85,B 0,C 180,E1 -7736.551,E2 -7736.551} C_VEL
LIN {X 0,Y 467.308,Z 872.366,A -85,B 0,C 180,E1 -7737.414,E2 -7737.414} C_VEL
LIN {X 0,Y 467.1,Z 873.858,A -85,B 0,C 180,E1 -7739.138,E2 -7739.138} C_VEL
LIN {X 0,Y 467.099,Z 874.02,A -85,B 0,C 180,E1 -7740,E2 -7740} C_VEL
LIN {X 0,Y 467.1,Z 873.768,A -85,B 0,C 180,E1 -7740.862,E2 -7740.862} C_VEL
LIN {X 0,Y 467.136,Z 872.053,A -85,B 0,C 180,E1 -7742.587,E2 -7742.587} C_VEL
LIN {X 0,Y 467.319,Z 868.686,A -85,B 0,C 180,E1 -7744.312,E2 -7744.312} C_VEL
LIN {X 0,Y 467.428,Z 865.014,A -85,B 0,C 180,E1 -7745.609,E2 -7745.609} C_VEL
LIN {X 0,Y 467.638,Z 860.212,A -85,B 0,C 180,E1 -7746.905,E2 -7746.905} C_VEL
LIN {X 0,Y 467.814,Z 855.301,A -85,B 0,C 180,E1 -7747.988,E2 -7747.988} C_VEL
LIN {X 0,Y 468.134,Z 848.055,A -85,B 0,C 180,E1 -7749.288,E2 -7749.288} C_VEL
LIN {X 0,Y 468.412,Z 840.553,A -85,B 0,C 180,E1 -7750.373,E2 -7750.373} C_VEL
LIN {X 0,Y 468.729,Z 833.527,A -85,B 0,C 180,E1 -7751.24,E2 -7751.24} C_VEL
LIN {X 0,Y 468.996,Z 825.22,A -85,B 0,C 180,E1 -7752.11,E2 -7752.11} C_VEL
LIN {X 0,Y 469.474,Z 814.136,A -85,B 0,C 180,E1 -7753.066,E2 -7753.066} C_VEL
LIN {X 0,Y 469.788,Z 803.964,A -85,B 0,C 180,E1 -7753.75,E2 -7753.75} C_VEL
LIN {X 0,Y 469.296,Z 800.678,A -85,B 0,C 180,E1 -7753.974,E2 -7753.974} C_VEL
LIN {X 0,Y 467.58,Z 794.24,A -85,B 0,C 180,E1 -7754.387,E2 -7754.387} C_VEL
LIN {X 0,Y 467.545,Z 794.249,A -85,B 0,C 180,E1 -7757.496,E2 -7757.496} C_VEL
LIN {X 0,Y 467.533,Z 794.24,A -85,B 0,C 180,E1 -7760.227,E2 -7760.227} C_VEL
LIN {X 0,Y 467.57,Z 794.242,A -85,B 0,C 180,E1 -7763.523,E2 -7763.523} C_VEL
LIN {X 0,Y 467.556,Z 794.243,A -85,B 0,C 180,E1 -7765.843,E2 -7765.843} C_VEL
LIN {X 0,Y 467.54,Z 794.239,A -85,B 0,C 180,E1 -7768.752,E2 -7768.752} C_VEL
LIN {X 0,Y 467.576,Z 794.242,A -85,B 0,C 180,E1 -7771.741,E2 -7771.741} C_VEL
LIN {X 0,Y 467.555,Z 794.238,A -85,B 0,C 180,E1 -7774.834,E2 -7774.834} C_VEL
LIN {X 0,Y 467.546,Z 794.245,A -85,B 0,C 180,E1 -7778.047,E2 -7778.047} C_VEL
LIN {X 0,Y 467.568,Z 794.238,A -85,B 0,C 180,E1 -7781.274,E2 -7781.274} C_VEL
LIN {X 0,Y 467.571,Z 794.237,A -85,B 0,C 180,E1 -7784.947,E2 -7784.947} C_VEL
LIN {X 0,Y 467.567,Z 794.239,A -85,B 0,C 180,E1 -7787.436,E2 -7787.436} C_VEL
LIN {X 0,Y 467.57,Z 794.244,A -85,B 0,C 180,E1 -7790.048,E2 -7790.048} C_VEL
LIN {X 0,Y 467.53,Z 794.241,A -85,B 0,C 180,E1 -7793.037,E2 -7793.037} C_VEL
LIN {X 0,Y 467.576,Z 794.245,A -85,B 0,C 180,E1 -7796.21,E2 -7796.21} C_VEL
LIN {X 0,Y 467.574,Z 794.235,A -85,B 0,C 180,E1 -7799.265,E2 -7799.265} C_VEL
LIN {X 0,Y 467.635,Z 794.233,A -85,B 0,C 180,E1 -7802.462,E2 -7802.462} C_VEL
LIN {X 0,Y 467.575,Z 794.233,A -85,B 0,C 180,E1 -7805.11,E2 -7805.11} C_VEL
LIN {X 0,Y 467.541,Z 794.245,A -85,B 0,C 180,E1 -7807.925,E2 -7807.925} C_VEL
LIN {X 0,Y 467.628,Z 794.24,A -85,B 0,C 180,E1 -7810.691,E2 -7810.691} C_VEL
LIN {X 0,Y 467.627,Z 794.235,A -85,B 0,C 180,E1 -7811.553,E2 -7811.553} C_VEL
LIN {X 0,Y 466.966,Z 794.321,A -85,B 0,C 180,E1 -7812.033,E2 -7812.033} C_VEL
LIN {X 0,Y 464.118,Z 794.676,A -85,B 0,C 180,E1 -7812.784,E2 -7812.784} C_VEL
LIN {X 0,Y 461.262,Z 795.029,A -85,B 0,C 180,E1 -7813.543,E2 -7813.543} C_VEL
LIN {X 0,Y 460.608,Z 795.112,A -85,B 0,C 180,E1 -7814.034,E2 -7814.034} C_VEL
LIN {X 0,Y 460.581,Z 795.112,A -85,B 0,C 180,E1 -7815.134,E2 -7815.134} C_VEL
LIN {X 0,Y 463.652,Z 806.163,A -85,B 0,C 180,E1 -7815.851,E2 -7815.851} C_VEL
LIN {X 0,Y 463.395,Z 816.681,A -85,B 0,C 180,E1 -7816.559,E2 -7816.559} C_VEL
LIN {X 0,Y 462.838,Z 827.839,A -85,B 0,C 180,E1 -7817.502,E2 -7817.502} C_VEL
LIN {X 0,Y 462.357,Z 838.195,A -85,B 0,C 180,E1 -7818.602,E2 -7818.602} C_VEL
LIN {X 0,Y 461.926,Z 846.575,A -85,B 0,C 180,E1 -7819.7,E2 -7819.7} C_VEL
LIN {X 0,Y 461.429,Z 854.701,A -85,B 0,C 180,E1 -7821.017,E2 -7821.017} C_VEL
LIN {X 0,Y 461.182,Z 860.239,A -85,B 0,C 180,E1 -7822.115,E2 -7822.115} C_VEL
LIN {X 0,Y 460.989,Z 865.622,A -85,B 0,C 180,E1 -7823.433,E2 -7823.433} C_VEL
LIN {X 0,Y 460.564,Z 869.883,A -85,B 0,C 180,E1 -7824.745,E2 -7824.745} C_VEL
LIN {X 0,Y 460.504,Z 872.108,A -85,B 0,C 180,E1 -7825.622,E2 -7825.622} C_VEL
LIN {X 0,Y 460.39,Z 873.93,A -85,B 0,C 180,E1 -7826.498,E2 -7826.498} C_VEL
LIN {X 0,Y 460.407,Z 875.291,A -85,B 0,C 180,E1 -7827.374,E2 -7827.374} C_VEL
LIN {X 0,Y 460.272,Z 876.279,A -85,B 0,C 180,E1 -7828.248,E2 -7828.248} C_VEL
LIN {X 0,Y 460.332,Z 877.098,A -85,B 0,C 180,E1 -7829.998,E2 -7829.998} C_VEL
LIN {X 0,Y 460.309,Z 876.922,A -85,B 0,C 180,E1 -7830.873,E2 -7830.873} C_VEL
LIN {X 0,Y 460.405,Z 875.411,A -85,B 0,C 180,E1 -7832.623,E2 -7832.623} C_VEL
LIN {X 0,Y 460.384,Z 874.104,A -85,B 0,C 180,E1 -7833.499,E2 -7833.499} C_VEL
LIN {X 0,Y 460.55,Z 871.302,A -85,B 0,C 180,E1 -7834.813,E2 -7834.813} C_VEL
LIN {X 0,Y 460.876,Z 867.484,A -85,B 0,C 180,E1 -7836.126,E2 -7836.126} C_VEL
LIN {X 0,Y 461.104,Z 862.449,A -85,B 0,C 180,E1 -7837.476,E2 -7837.476} C_VEL
LIN {X 0,Y 461.376,Z 856.412,A -85,B 0,C 180,E1 -7838.76,E2 -7838.76} C_VEL
LIN {X 0,Y 461.838,Z 848.65,A -85,B 0,C 180,E1 -7840.077,E2 -7840.077} C_VEL
LIN {X 0,Y 462.266,Z 840.729,A -85,B 0,C 180,E1 -7841.175,E2 -7841.175} C_VEL
LIN {X 0,Y 462.714,Z 831.051,A -85,B 0,C 180,E1 -7842.275,E2 -7842.275} C_VEL
LIN {X 0,Y 463.13,Z 821.509,A -85,B 0,C 180,E1 -7843.155,E2 -7843.155} C_VEL
LIN {X 0,Y 463.528,Z 810.286,A -85,B 0,C 180,E1 -7843.982,E2 -7843.982} C_VEL
LIN {X 0,Y 463.624,Z 805.876,A -85,B 0,C 180,E1 -7844.259,E2 -7844.259} C_VEL
LIN {X 0,Y 460.574,Z 795.115,A -85,B 0,C 180,E1 -7844.976,E2 -7844.976} C_VEL
LIN {X 0,Y 460.559,Z 795.119,A -85,B 0,C 180,E1 -7847.768,E2 -7847.768} C_VEL
LIN {X 0,Y 460.55,Z 795.113,A -85,B 0,C 180,E1 -7850.545,E2 -7850.545} C_VEL
LIN {X 0,Y 460.535,Z 795.121,A -85,B 0,C 180,E1 -7853.704,E2 -7853.704} C_VEL
LIN {X 0,Y 460.559,Z 795.116,A -85,B 0,C 180,E1 -7856.263,E2 -7856.263} C_VEL
LIN {X 0,Y 460.536,Z 795.116,A -85,B 0,C 180,E1 -7859.229,E2 -7859.229} C_VEL
LIN {X 0,Y 460.527,Z 795.121,A -85,B 0,C 180,E1 -7862.282,E2 -7862.282} C_VEL
LIN {X 0,Y 460.506,Z 795.12,A -85,B 0,C 180,E1 -7865.444,E2 -7865.444} C_VEL
LIN {X 0,Y 460.55,Z 795.114,A -85,B 0,C 180,E1 -7868.898,E2 -7868.898} C_VEL
LIN {X 0,Y 460.539,Z 795.121,A -85,B 0,C 180,E1 -7872.177,E2 -7872.177} C_VEL
LIN {X 0,Y 460.512,Z 795.117,A -85,B 0,C 180,E1 -7875.41,E2 -7875.41} C_VEL
LIN {X 0,Y 460.534,Z 795.12,A -85,B 0,C 180,E1 -7878.394,E2 -7878.394} C_VEL
LIN {X 0,Y 460.535,Z 795.112,A -85,B 0,C 180,E1 -7881.268,E2 -7881.268} C_VEL
LIN {X 0,Y 460.5,Z 795.125,A -85,B 0,C 180,E1 -7884.553,E2 -7884.553} C_VEL
LIN {X 0,Y 460.519,Z 795.116,A -85,B 0,C 180,E1 -7887.714,E2 -7887.714} C_VEL
LIN {X 0,Y 460.532,Z 795.12,A -85,B 0,C 180,E1 -7890.768,E2 -7890.768} C_VEL
LIN {X 0,Y 460.553,Z 795.11,A -85,B 0,C 180,E1 -7893.734,E2 -7893.734} C_VEL
LIN {X 0,Y 460.53,Z 795.119,A -85,B 0,C 180,E1 -7896.623,E2 -7896.623} C_VEL
LIN {X 0,Y 460.535,Z 795.115,A -85,B 0,C 180,E1 -7899.452,E2 -7899.452} C_VEL
LIN {X 0,Y 460.542,Z 795.113,A -85,B 0,C 180,E1 -7902.229,E2 -7902.229} C_VEL
LIN {X 0,Y 460.548,Z 795.115,A -85,B 0,C 180,E1 -7904.964,E2 -7904.964} C_VEL
LIN {X 0,Y 460.613,Z 795.108,A -85,B 0,C 180,E1 -7907.666,E2 -7907.666} C_VEL
LIN {X 0,Y 460.613,Z 795.108,A -85,B 0,C 180,E1 -7911.223,E2 -7911.223} C_VEL
LIN {X 0,Y 460.684,Z 795.1,A -85,B 0,C 180,E1 -7913.87,E2 -7913.87} C_VEL
LIN {X 0,Y 460.807,Z 795.085,A -85,B 0,C 180,E1 -7917.377,E2 -7917.377} C_VEL
LIN {X 0,Y 460.833,Z 795.081,A -85,B 0,C 180,E1 -7920,E2 -7920} C_VEL
LIN {X 0,Y 460.782,Z 795.085,A -85,B 0,C 180,E1 -7922.623,E2 -7922.623} C_VEL
LIN {X 0,Y 460.666,Z 795.1,A -85,B 0,C 180,E1 -7926.13,E2 -7926.13} C_VEL
LIN {X 0,Y 460.61,Z 795.105,A -85,B 0,C 180,E1 -7928.776,E2 -7928.776} C_VEL
LIN {X 0,Y 460.617,Z 795.102,A -85,B 0,C 180,E1 -7932.457,E2 -7932.457} C_VEL
LIN {X 0,Y 460.583,Z 795.116,A -85,B 0,C 180,E1 -7935.998,E2 -7935.998} C_VEL
LIN {X 0,Y 460.55,Z 795.117,A -85,B 0,C 180,E1 -7939.616,E2 -7939.616} C_VEL
LIN {X 0,Y 460.493,Z 795.123,A -85,B 0,C 180,E1 -7942.43,E2 -7942.43} C_VEL
LIN {X 0,Y 460.529,Z 795.119,A -85,B 0,C 180,E1 -7945.797,E2 -7945.797} C_VEL
LIN {X 0,Y 460.51,Z 795.124,A -85,B 0,C 180,E1 -7948.236,E2 -7948.236} C_VEL
LIN {X 0,Y 460.505,Z 795.119,A -85,B 0,C 180,E1 -7951.284,E2 -7951.284} C_VEL
LIN {X 0,Y 460.506,Z 795.124,A -85,B 0,C 180,E1 -7954.505,E2 -7954.505} C_VEL
LIN {X 0,Y 460.471,Z 795.124,A -85,B 0,C 180,E1 -7957.626,E2 -7957.626} C_VEL
LIN {X 0,Y 460.502,Z 795.121,A -85,B 0,C 180,E1 -7961.015,E2 -7961.015} C_VEL
LIN {X 0,Y 460.498,Z 795.122,A -85,B 0,C 180,E1 -7964.591,E2 -7964.591} C_VEL
LIN {X 0,Y 460.462,Z 795.129,A -85,B 0,C 180,E1 -7967.815,E2 -7967.815} C_VEL
LIN {X 0,Y 460.533,Z 795.253,A -85,B 0,C 180,E1 -7968.992,E2 -7968.992} C_VEL
LIN {X 0,Y 462.7,Z 806.285,A -85,B 0,C 180,E1 -7972.17,E2 -7972.17} C_VEL
LIN {X 0,Y 463.441,Z 811.141,A -85,B 0,C 180,E1 -7973.489,E2 -7973.489} C_VEL
LIN {X 0,Y 463.107,Z 820.507,A -85,B 0,C 180,E1 -7975.843,E2 -7975.843} C_VEL
LIN {X 0,Y 462.609,Z 833.143,A -85,B 0,C 180,E1 -7978.903,E2 -7978.903} C_VEL
LIN {X 0,Y 461.983,Z 848.953,A -85,B 0,C 180,E1 -7982.608,E2 -7982.608} C_VEL
LIN {X 0,Y 461.518,Z 862.5,A -85,B 0,C 180,E1 -7985.725,E2 -7985.725} C_VEL
LIN {X 0,Y 461.01,Z 877.925,A -85,B 0,C 180,E1 -7989.243,E2 -7989.243} C_VEL
LIN {X 0,Y 460.647,Z 892.085,A -85,B 0,C 180,E1 -7992.465,E2 -7992.465} C_VEL
LIN {X 0,Y 460.422,Z 900.141,A -85,B 0,C 180,E1 -7994.31,E2 -7994.31} C_VEL
LIN {X 0,Y 461.836,Z 914.191,A -85,B 0,C 180,E1 -7994.699,E2 -7994.699} C_VEL
LIN {X 0,Y 462.982,Z 924.39,A -85,B 0,C 180,E1 -7995.103,E2 -7995.103} C_VEL
LIN {X 0,Y 462.553,Z 936.844,A -85,B 0,C 180,E1 -7995.708,E2 -7995.708} C_VEL
LIN {X 0,Y 462.002,Z 948.843,A -85,B 0,C 180,E1 -7996.476,E2 -7996.476} C_VEL
LIN {X 0,Y 461.516,Z 959.638,A -85,B 0,C 180,E1 -7997.359,E2 -7997.359} C_VEL
LIN {X 0,Y 460.982,Z 969.486,A -85,B 0,C 180,E1 -7998.348,E2 -7998.348} C_VEL
LIN {X 0,Y 460.583,Z 978.51,A -85,B 0,C 180,E1 -7999.451,E2 -7999.451} C_VEL
LIN {X 0,Y 460.246,Z 987.34,A -85,B 0,C 180,E1 -8000.775,E2 -8000.775} C_VEL
LIN {X 0,Y 459.995,Z 994.412,A -85,B 0,C 180,E1 -8002.098,E2 -8002.098} C_VEL
LIN {X 0,Y 459.877,Z 999.988,A -85,B 0,C 180,E1 -8003.392,E2 -8003.392} C_VEL
LIN {X 0,Y 459.791,Z 1004.564,A -85,B 0,C 180,E1 -8004.74,E2 -8004.74} C_VEL
LIN {X 0,Y 459.765,Z 1006.934,A -85,B 0,C 180,E1 -8005.618,E2 -8005.618} C_VEL
LIN {X 0,Y 459.8,Z 1008.864,A -85,B 0,C 180,E1 -8006.496,E2 -8006.496} C_VEL
LIN {X 0,Y 459.734,Z 1010.297,A -85,B 0,C 180,E1 -8007.373,E2 -8007.373} C_VEL
LIN {X 0,Y 459.729,Z 1011.324,A -85,B 0,C 180,E1 -8008.25,E2 -8008.25} C_VEL
LIN {X 0,Y 459.695,Z 1011.946,A -85,B 0,C 180,E1 -8009.126,E2 -8009.126} C_VEL
LIN {X 0,Y 459.685,Z 1012.167,A -85,B 0,C 180,E1 -8010.002,E2 -8010.002} C_VEL
LIN {X 0,Y 459.695,Z 1011.944,A -85,B 0,C 180,E1 -8010.878,E2 -8010.878} C_VEL
LIN {X 0,Y 459.729,Z 1011.32,A -85,B 0,C 180,E1 -8011.754,E2 -8011.754} C_VEL
LIN {X 0,Y 459.735,Z 1010.29,A -85,B 0,C 180,E1 -8012.63,E2 -8012.63} C_VEL
LIN {X 0,Y 459.801,Z 1008.854,A -85,B 0,C 180,E1 -8013.507,E2 -8013.507} C_VEL
LIN {X 0,Y 459.788,Z 1005.821,A -85,B 0,C 180,E1 -8014.824,E2 -8014.824} C_VEL
LIN {X 0,Y 459.878,Z 1001.733,A -85,B 0,C 180,E1 -8016.143,E2 -8016.143} C_VEL
LIN {X 0,Y 459.968,Z 995.435,A -85,B 0,C 180,E1 -8017.685,E2 -8017.685} C_VEL
LIN {X 0,Y 460.183,Z 988.586,A -85,B 0,C 180,E1 -8019.008,E2 -8019.008} C_VEL
LIN {X 0,Y 460.527,Z 980.114,A -85,B 0,C 180,E1 -8020.331,E2 -8020.331} C_VEL
LIN {X 0,Y 460.995,Z 971.46,A -85,B 0,C 180,E1 -8021.432,E2 -8021.432} C_VEL
LIN {X 0,Y 461.519,Z 961.33,A -85,B 0,C 180,E1 -8022.484,E2 -8022.484} C_VEL
LIN {X 0,Y 461.913,Z 950.243,A -85,B 0,C 180,E1 -8023.418,E2 -8023.418} C_VEL
LIN {X 0,Y 462.461,Z 938.74,A -85,B 0,C 180,E1 -8024.186,E2 -8024.186} C_VEL
LIN {X 0,Y 462.893,Z 926.947,A -85,B 0,C 180,E1 -8024.79,E2 -8024.79} C_VEL
LIN {X 0,Y 462.796,Z 921.19,A -85,B 0,C 180,E1 -8025.033,E2 -8025.033} C_VEL
LIN {X 0,Y 461.318,Z 909.05,A -85,B 0,C 180,E1 -8025.464,E2 -8025.464} C_VEL
LIN {X 0,Y 460.428,Z 900.154,A -85,B 0,C 180,E1 -8025.693,E2 -8025.693} C_VEL
LIN {X 0,Y 460.794,Z 887.044,A -85,B 0,C 180,E1 -8028.682,E2 -8028.682} C_VEL
LIN {X 0,Y 461.148,Z 872.701,A -85,B 0,C 180,E1 -8031.951,E2 -8031.951} C_VEL
LIN {X 0,Y 461.605,Z 860.409,A -85,B 0,C 180,E1 -8034.753,E2 -8034.753} C_VEL
LIN {X 0,Y 462.062,Z 846.925,A -85,B 0,C 180,E1 -8037.86,E2 -8037.86} C_VEL
LIN {X 0,Y 462.647,Z 831.812,A -85,B 0,C 180,E1 -8041.412,E2 -8041.412} C_VEL
LIN {X 0,Y 463.211,Z 818.804,A -85,B 0,C 180,E1 -8044.576,E2 -8044.576} C_VEL
LIN {X 0,Y 463.419,Z 811.138,A -85,B 0,C 180,E1 -8046.508,E2 -8046.508} C_VEL
LIN {X 0,Y 462.463,Z 805.156,A -85,B 0,C 180,E1 -8048.14,E2 -8048.14} C_VEL
LIN {X 0,Y 460.511,Z 795.123,A -85,B 0,C 180,E1 -8051.074,E2 -8051.074} C_VEL
LIN {X 0,Y 460.488,Z 795.125,A -85,B 0,C 180,E1 -8054.593,E2 -8054.593} C_VEL
LIN {X 0,Y 460.498,Z 795.122,A -85,B 0,C 180,E1 -8058.404,E2 -8058.404} C_VEL
LIN {X 0,Y 460.492,Z 795.124,A -85,B 0,C 180,E1 -8061.263,E2 -8061.263} C_VEL
LIN {X 0,Y 460.465,Z 795.125,A -85,B 0,C 180,E1 -8064.55,E2 -8064.55} C_VEL
LIN {X 0,Y 460.502,Z 795.124,A -85,B 0,C 180,E1 -8067.713,E2 -8067.713} C_VEL
LIN {X 0,Y 460.5,Z 795.121,A -85,B 0,C 180,E1 -8070.766,E2 -8070.766} C_VEL
LIN {X 0,Y 460.464,Z 795.128,A -85,B 0,C 180,E1 -8073.729,E2 -8073.729} C_VEL
LIN {X 0,Y 460.524,Z 795.12,A -85,B 0,C 180,E1 -8076.623,E2 -8076.623} C_VEL
LIN {X 0,Y 460.48,Z 795.125,A -85,B 0,C 180,E1 -8079.449,E2 -8079.449} C_VEL
LIN {X 0,Y 460.498,Z 795.128,A -85,B 0,C 180,E1 -8082.228,E2 -8082.228} C_VEL
LIN {X 0,Y 460.567,Z 795.287,A -85,B 0,C 180,E1 -8085.332,E2 -8085.332} C_VEL
LIN {X 0,Y 463.183,Z 804.644,A -85,B 0,C 180,E1 -8085.95,E2 -8085.95} C_VEL
LIN {X 0,Y 462.968,Z 815.292,A -85,B 0,C 180,E1 -8086.672,E2 -8086.672} C_VEL
LIN {X 0,Y 462.585,Z 825.159,A -85,B 0,C 180,E1 -8087.497,E2 -8087.497} C_VEL
LIN {X 0,Y 462.218,Z 833.845,A -85,B 0,C 180,E1 -8088.377,E2 -8088.377} C_VEL
LIN {X 0,Y 461.792,Z 842.894,A -85,B 0,C 180,E1 -8089.477,E2 -8089.477} C_VEL
LIN {X 0,Y 461.431,Z 850.09,A -85,B 0,C 180,E1 -8090.576,E2 -8090.576} C_VEL
LIN {X 0,Y 461.137,Z 855.064,A -85,B 0,C 180,E1 -8091.454,E2 -8091.454} C_VEL
LIN {X 0,Y 460.996,Z 859.738,A -85,B 0,C 180,E1 -8092.421,E2 -8092.421} C_VEL
LIN {X 0,Y 460.717,Z 865.38,A -85,B 0,C 180,E1 -8093.87,E2 -8093.87} C_VEL
LIN {X 0,Y 460.436,Z 868.133,A -85,B 0,C 180,E1 -8094.745,E2 -8094.745} C_VEL
LIN {X 0,Y 460.286,Z 872.039,A -85,B 0,C 180,E1 -8096.499,E2 -8096.499} C_VEL
LIN {X 0,Y 460.305,Z 873.466,A -85,B 0,C 180,E1 -8097.375,E2 -8097.375} C_VEL
LIN {X 0,Y 460.111,Z 874.936,A -85,B 0,C 180,E1 -8099.125,E2 -8099.125} C_VEL
LIN {X 0,Y 460.105,Z 875.087,A -85,B 0,C 180,E1 -8100,E2 -8100} C_VEL
LIN {X 0,Y 460.084,Z 874.824,A -85,B 0,C 180,E1 -8100.875,E2 -8100.875} C_VEL
LIN {X 0,Y 460.119,Z 873.082,A -85,B 0,C 180,E1 -8102.626,E2 -8102.626} C_VEL
LIN {X 0,Y 460.309,Z 869.672,A -85,B 0,C 180,E1 -8104.378,E2 -8104.378} C_VEL
LIN {X 0,Y 460.435,Z 865.966,A -85,B 0,C 180,E1 -8105.694,E2 -8105.694} C_VEL
LIN {X 0,Y 460.66,Z 861.126,A -85,B 0,C 180,E1 -8107.011,E2 -8107.011} C_VEL
LIN {X 0,Y 460.855,Z 856.179,A -85,B 0,C 180,E1 -8108.109,E2 -8108.109} C_VEL
LIN {X 0,Y 461.195,Z 848.892,A -85,B 0,C 180,E1 -8109.429,E2 -8109.429} C_VEL
LIN {X 0,Y 461.491,Z 841.338,A -85,B 0,C 180,E1 -8110.53,E2 -8110.53} C_VEL
LIN {X 0,Y 461.821,Z 834.264,A -85,B 0,C 180,E1 -8111.41,E2 -8111.41} C_VEL
LIN {X 0,Y 462.103,Z 825.902,A -85,B 0,C 180,E1 -8112.294,E2 -8112.294} C_VEL
LIN {X 0,Y 462.573,Z 815.886,A -85,B 0,C 180,E1 -8113.174,E2 -8113.174} C_VEL
LIN {X 0,Y 462.885,Z 806.135,A -85,B 0,C 180,E1 -8113.856,E2 -8113.856} C_VEL
LIN {X 0,Y 462.628,Z 802.964,A -85,B 0,C 180,E1 -8114.068,E2 -8114.068} C_VEL
LIN {X 0,Y 460.55,Z 795.116,A -85,B 0,C 180,E1 -8114.584,E2 -8114.584} C_VEL
LIN {X 0,Y 460.498,Z 795.125,A -85,B 0,C 180,E1 -8117.772,E2 -8117.772} C_VEL
LIN {X 0,Y 460.48,Z 795.117,A -85,B 0,C 180,E1 -8120.551,E2 -8120.551} C_VEL
LIN {X 0,Y 460.508,Z 795.124,A -85,B 0,C 180,E1 -8123.695,E2 -8123.695} C_VEL
LIN {X 0,Y 460.483,Z 795.118,A -85,B 0,C 180,E1 -8126.27,E2 -8126.27} C_VEL
LIN {X 0,Y 460.518,Z 795.116,A -85,B 0,C 180,E1 -8129.233,E2 -8129.233} C_VEL
LIN {X 0,Y 460.527,Z 795.112,A -85,B 0,C 180,E1 -8132.285,E2 -8132.285} C_VEL
LIN {X 0,Y 460.505,Z 795.119,A -85,B 0,C 180,E1 -8135.446,E2 -8135.446} C_VEL
LIN {X 0,Y 460.497,Z 795.117,A -85,B 0,C 180,E1 -8138.889,E2 -8138.889} C_VEL
LIN {X 0,Y 460.51,Z 795.12,A -85,B 0,C 180,E1 -8141.598,E2 -8141.598} C_VEL
LIN {X 0,Y 460.518,Z 795.118,A -85,B 0,C 180,E1 -8144.589,E2 -8144.589} C_VEL
LIN {X 0,Y 460.509,Z 795.122,A -85,B 0,C 180,E1 -8147.816,E2 -8147.816} C_VEL
LIN {X 0,Y 460.52,Z 795.122,A -85,B 0,C 180,E1 -8150.135,E2 -8150.135} C_VEL
LIN {X 0,Y 460.479,Z 795.12,A -85,B 0,C 180,E1 -8153.469,E2 -8153.469} C_VEL
LIN {X 0,Y 460.526,Z 795.117,A -85,B 0,C 180,E1 -8156.674,E2 -8156.674} C_VEL
LIN {X 0,Y 460.516,Z 795.117,A -85,B 0,C 180,E1 -8159.759,E2 -8159.759} C_VEL
LIN {X 0,Y 460.564,Z 795.111,A -85,B 0,C 180,E1 -8162.754,E2 -8162.754} C_VEL
LIN {X 0,Y 460.528,Z 795.111,A -85,B 0,C 180,E1 -8165.666,E2 -8165.666} C_VEL
LIN {X 0,Y 460.528,Z 795.123,A -85,B 0,C 180,E1 -8168.577,E2 -8168.577} C_VEL
LIN {X 0,Y 460.57,Z 795.115,A -85,B 0,C 180,E1 -8171.545,E2 -8171.545} C_VEL
LIN {X 0,Y 460.608,Z 795.112,A -85,B 0,C 180,E1 -8174.034,E2 -8174.034} C_VEL
LIN {X 0,Y 460.446,Z 795.952,A -85,B 0,C 180,E1 -8174.483,E2 -8174.483} C_VEL
LIN {X 0,Y 460.017,Z 797.972,A -85,B 0,C 180,E1 -8174.878,E2 -8174.878} C_VEL
LIN {X 0,Y 459.103,Z 802.333,A -85,B 0,C 180,E1 -8175.362,E2 -8175.362} C_VEL
LIN {X 0,Y 458.028,Z 808.201,A -85,B 0,C 180,E1 -8175.748,E2 -8175.748} C_VEL
LIN {X 0,Y 457.346,Z 812.231,A -85,B 0,C 180,E1 -8175.984,E2 -8175.984} C_VEL
LIN {X 0,Y 456.473,Z 819.542,A -85,B 0,C 180,E1 -8176.498,E2 -8176.498} C_VEL
LIN {X 0,Y 455.931,Z 830.027,A -85,B 0,C 180,E1 -8177.423,E2 -8177.423} C_VEL
LIN {X 0,Y 455.475,Z 839.23,A -85,B 0,C 180,E1 -8178.427,E2 -8178.427} C_VEL
LIN {X 0,Y 455.019,Z 847.609,A -85,B 0,C 180,E1 -8179.542,E2 -8179.542} C_VEL
LIN {X 0,Y 454.495,Z 855.734,A -85,B 0,C 180,E1 -8180.879,E2 -8180.879} C_VEL
LIN {X 0,Y 454.115,Z 863.092,A -85,B 0,C 180,E1 -8182.407,E2 -8182.407} C_VEL
LIN {X 0,Y 453.904,Z 868.216,A -85,B 0,C 180,E1 -8183.776,E2 -8183.776} C_VEL
LIN {X 0,Y 453.556,Z 872.104,A -85,B 0,C 180,E1 -8185.11,E2 -8185.11} C_VEL
LIN {X 0,Y 453.379,Z 874.963,A -85,B 0,C 180,E1 -8186.444,E2 -8186.444} C_VEL
LIN {X 0,Y 453.395,Z 876.322,A -85,B 0,C 180,E1 -8187.333,E2 -8187.333} C_VEL
LIN {X 0,Y 453.256,Z 877.31,A -85,B 0,C 180,E1 -8188.221,E2 -8188.221} C_VEL
LIN {X 0,Y 453.316,Z 878.128,A -85,B 0,C 180,E1 -8189.998,E2 -8189.998} C_VEL
LIN {X 0,Y 453.298,Z 877.951,A -85,B 0,C 180,E1 -8190.887,E2 -8190.887} C_VEL
LIN {X 0,Y 453.393,Z 876.441,A -85,B 0,C 180,E1 -8192.664,E2 -8192.664} C_VEL
LIN {X 0,Y 453.372,Z 875.134,A -85,B 0,C 180,E1 -8193.553,E2 -8193.553} C_VEL
LIN {X 0,Y 453.549,Z 872.332,A -85,B 0,C 180,E1 -8194.887,E2 -8194.887} C_VEL
LIN {X 0,Y 453.902,Z 868.513,A -85,B 0,C 180,E1 -8196.221,E2 -8196.221} C_VEL
LIN {X 0,Y 454.143,Z 863.451,A -85,B 0,C 180,E1 -8197.598,E2 -8197.598} C_VEL
LIN {X 0,Y 454.433,Z 857.441,A -85,B 0,C 180,E1 -8198.895,E2 -8198.895} C_VEL
LIN {X 0,Y 454.926,Z 849.678,A -85,B 0,C 180,E1 -8200.232,E2 -8200.232} C_VEL
LIN {X 0,Y 455.377,Z 841.757,A -85,B 0,C 180,E1 -8201.347,E2 -8201.347} C_VEL
LIN {X 0,Y 455.852,Z 832.077,A -85,B 0,C 180,E1 -8202.463,E2 -8202.463} C_VEL
LIN {X 0,Y 456.299,Z 822.534,A -85,B 0,C 180,E1 -8203.356,E2 -8203.356} C_VEL
LIN {X 0,Y 456.714,Z 811.297,A -85,B 0,C 180,E1 -8204.196,E2 -8204.196} C_VEL
LIN {X 0,Y 456.691,Z 806.919,A -85,B 0,C 180,E1 -8204.48,E2 -8204.48} C_VEL
LIN {X 0,Y 453.525,Z 795.993,A -85,B 0,C 180,E1 -8205.215,E2 -8205.215} C_VEL
LIN {X 0,Y 453.511,Z 795.995,A -85,B 0,C 180,E1 -8208.053,E2 -8208.053} C_VEL
LIN {X 0,Y 453.481,Z 795.993,A -85,B 0,C 180,E1 -8210.88,E2 -8210.88} C_VEL
LIN {X 0,Y 453.497,Z 795.998,A -85,B 0,C 180,E1 -8213.887,E2 -8213.887} C_VEL
LIN {X 0,Y 453.505,Z 795.991,A -85,B 0,C 180,E1 -8216.704,E2 -8216.704} C_VEL
LIN {X 0,Y 453.471,Z 796,A -85,B 0,C 180,E1 -8219.73,E2 -8219.73} C_VEL
LIN {X 0,Y 453.484,Z 795.994,A -85,B 0,C 180,E1 -8223.187,E2 -8223.187} C_VEL
LIN {X 0,Y 453.448,Z 796.004,A -85,B 0,C 180,E1 -8226.298,E2 -8226.298} C_VEL
LIN {X 0,Y 453.52,Z 795.989,A -85,B 0,C 180,E1 -8229.444,E2 -8229.444} C_VEL
LIN {X 0,Y 453.482,Z 795.994,A -85,B 0,C 180,E1 -8232.99,E2 -8232.99} C_VEL
LIN {X 0,Y 453.467,Z 795.997,A -85,B 0,C 180,E1 -8235.779,E2 -8235.779} C_VEL
LIN {X 0,Y 453.485,Z 795.995,A -85,B 0,C 180,E1 -8238.21,E2 -8238.21} C_VEL
LIN {X 0,Y 453.521,Z 795.99,A -85,B 0,C 180,E1 -8240.786,E2 -8240.786} C_VEL
LIN {X 0,Y 453.444,Z 795.998,A -85,B 0,C 180,E1 -8243.916,E2 -8243.916} C_VEL
LIN {X 0,Y 453.469,Z 795.997,A -85,B 0,C 180,E1 -8247.15,E2 -8247.15} C_VEL
LIN {X 0,Y 453.5,Z 795.99,A -85,B 0,C 180,E1 -8250.27,E2 -8250.27} C_VEL
LIN {X 0,Y 453.499,Z 795.991,A -85,B 0,C 180,E1 -8253.293,E2 -8253.293} C_VEL
LIN {X 0,Y 453.488,Z 795.992,A -85,B 0,C 180,E1 -8256.238,E2 -8256.238} C_VEL
LIN {X 0,Y 453.466,Z 795.999,A -85,B 0,C 180,E1 -8259.117,E2 -8259.117} C_VEL
LIN {X 0,Y 453.494,Z 795.991,A -85,B 0,C 180,E1 -8261.944,E2 -8261.944} C_VEL
LIN {X 0,Y 453.523,Z 795.988,A -85,B 0,C 180,E1 -8264.726,E2 -8264.726} C_VEL
LIN {X 0,Y 453.585,Z 795.985,A -85,B 0,C 180,E1 -8267.472,E2 -8267.472} C_VEL
LIN {X 0,Y 453.577,Z 795.984,A -85,B 0,C 180,E1 -8271.086,E2 -8271.086} C_VEL
LIN {X 0,Y 453.652,Z 795.977,A -85,B 0,C 180,E1 -8273.774,E2 -8273.774} C_VEL
LIN {X 0,Y 453.747,Z 795.964,A -85,B 0,C 180,E1 -8277.337,E2 -8277.337} C_VEL
LIN {X 0,Y 453.803,Z 795.957,A -85,B 0,C 180,E1 -8280,E2 -8280} C_VEL
LIN {X 0,Y 453.726,Z 795.964,A -85,B 0,C 180,E1 -8282.663,E2 -8282.663} C_VEL
LIN {X 0,Y 453.632,Z 795.975,A -85,B 0,C 180,E1 -8286.226,E2 -8286.226} C_VEL
LIN {X 0,Y 453.574,Z 795.982,A -85,B 0,C 180,E1 -8288.914,E2 -8288.914} C_VEL
LIN {X 0,Y 453.584,Z 795.978,A -85,B 0,C 180,E1 -8292.551,E2 -8292.551} C_VEL
LIN {X 0,Y 453.527,Z 795.993,A -85,B 0,C 180,E1 -8296.197,E2 -8296.197} C_VEL
LIN {X 0,Y 453.499,Z 795.992,A -85,B 0,C 180,E1 -8299.04,E2 -8299.04} C_VEL
LIN {X 0,Y 453.459,Z 796.003,A -85,B 0,C 180,E1 -8301.837,E2 -8301.837} C_VEL
LIN {X 0,Y 453.478,Z 795.994,A -85,B 0,C 180,E1 -8304.737,E2 -8304.737} C_VEL
LIN {X 0,Y 453.474,Z 795.997,A -85,B 0,C 180,E1 -8307.951,E2 -8307.951} C_VEL
LIN {X 0,Y 453.46,Z 795.999,A -85,B 0,C 180,E1 -8310.761,E2 -8310.761} C_VEL
LIN {X 0,Y 453.452,Z 796.001,A -85,B 0,C 180,E1 -8313.915,E2 -8313.915} C_VEL
LIN {X 0,Y 453.424,Z 796.002,A -85,B 0,C 180,E1 -8317.193,E2 -8317.193} C_VEL
LIN {X 0,Y 453.456,Z 796.004,A -85,B 0,C 180,E1 -8320.613,E2 -8320.613} C_VEL
LIN {X 0,Y 453.446,Z 796.002,A -85,B 0,C 180,E1 -8324.224,E2 -8324.224} C_VEL
LIN {X 0,Y 453.404,Z 796.007,A -85,B 0,C 180,E1 -8327.001,E2 -8327.001} C_VEL
LIN {X 0,Y 453.468,Z 796.035,A -85,B 0,C 180,E1 -8328.656,E2 -8328.656} C_VEL
LIN {X 0,Y 455.651,Z 807.093,A -85,B 0,C 180,E1 -8331.908,E2 -8331.908} C_VEL
LIN {X 0,Y 456.476,Z 811.676,A -85,B 0,C 180,E1 -8333.188,E2 -8333.188} C_VEL
LIN {X 0,Y 456.319,Z 818.622,A -85,B 0,C 180,E1 -8334.981,E2 -8334.981} C_VEL
LIN {X 0,Y 455.668,Z 832.304,A -85,B 0,C 180,E1 -8338.375,E2 -8338.375} C_VEL
LIN {X 0,Y 455.058,Z 847.585,A -85,B 0,C 180,E1 -8342.036,E2 -8342.036} C_VEL
LIN {X 0,Y 454.532,Z 861.614,A -85,B 0,C 180,E1 -8345.327,E2 -8345.327} C_VEL
LIN {X 0,Y 454.064,Z 874.113,A -85,B 0,C 180,E1 -8348.231,E2 -8348.231} C_VEL
LIN {X 0,Y 453.66,Z 889.135,A -85,B 0,C 180,E1 -8351.719,E2 -8351.719} C_VEL
LIN {X 0,Y 453.352,Z 899.166,A -85,B 0,C 180,E1 -8354.056,E2 -8354.056} C_VEL
LIN {X 0,Y 454.892,Z 914.7,A -85,B 0,C 180,E1 -8354.508,E2 -8354.508} C_VEL
LIN {X 0,Y 456.03,Z 924.65,A -85,B 0,C 180,E1 -8354.928,E2 -8354.928} C_VEL
LIN {X 0,Y 455.629,Z 935.794,A -85,B 0,C 180,E1 -8355.486,E2 -8355.486} C_VEL
LIN {X 0,Y 455.01,Z 947.787,A -85,B 0,C 180,E1 -8356.264,E2 -8356.264} C_VEL
LIN {X 0,Y 454.474,Z 959.26,A -85,B 0,C 180,E1 -8357.224,E2 -8357.224} C_VEL
LIN {X 0,Y 453.973,Z 968.435,A -85,B 0,C 180,E1 -8358.165,E2 -8358.165} C_VEL
LIN {X 0,Y 453.562,Z 977.461,A -85,B 0,C 180,E1 -8359.286,E2 -8359.286} C_VEL
LIN {X 0,Y 453.216,Z 986.294,A -85,B 0,C 180,E1 -8360.631,E2 -8360.631} C_VEL
LIN {X 0,Y 452.946,Z 993.367,A -85,B 0,C 180,E1 -8361.974,E2 -8361.974} C_VEL
LIN {X 0,Y 452.821,Z 999.254,A -85,B 0,C 180,E1 -8363.371,E2 -8363.371} C_VEL
LIN {X 0,Y 452.738,Z 1003.524,A -85,B 0,C 180,E1 -8364.657,E2 -8364.657} C_VEL
LIN {X 0,Y 452.727,Z 1005.897,A -85,B 0,C 180,E1 -8365.55,E2 -8365.55} C_VEL
LIN {X 0,Y 452.762,Z 1007.828,A -85,B 0,C 180,E1 -8366.442,E2 -8366.442} C_VEL
LIN {X 0,Y 452.7,Z 1009.263,A -85,B 0,C 180,E1 -8367.332,E2 -8367.332} C_VEL
LIN {X 0,Y 452.696,Z 1010.291,A -85,B 0,C 180,E1 -8368.222,E2 -8368.222} C_VEL
LIN {X 0,Y 452.669,Z 1010.914,A -85,B 0,C 180,E1 -8369.112,E2 -8369.112} C_VEL
LIN {X 0,Y 452.661,Z 1011.136,A -85,B 0,C 180,E1 -8370.002,E2 -8370.002} C_VEL
LIN {X 0,Y 452.669,Z 1010.912,A -85,B 0,C 180,E1 -8370.891,E2 -8370.891} C_VEL
LIN {X 0,Y 452.697,Z 1010.287,A -85,B 0,C 180,E1 -8371.781,E2 -8371.781} C_VEL
LIN {X 0,Y 452.7,Z 1009.256,A -85,B 0,C 180,E1 -8372.671,E2 -8372.671} C_VEL
LIN {X 0,Y 452.763,Z 1007.819,A -85,B 0,C 180,E1 -8373.561,E2 -8373.561} C_VEL
LIN {X 0,Y 452.751,Z 1004.785,A -85,B 0,C 180,E1 -8374.899,E2 -8374.899} C_VEL
LIN {X 0,Y 452.8,Z 1000.688,A -85,B 0,C 180,E1 -8376.239,E2 -8376.239} C_VEL
LIN {X 0,Y 452.906,Z 994.389,A -85,B 0,C 180,E1 -8377.805,E2 -8377.805} C_VEL
LIN {X 0,Y 453.134,Z 987.538,A -85,B 0,C 180,E1 -8379.149,E2 -8379.149} C_VEL
LIN {X 0,Y 453.466,Z 979.06,A -85,B 0,C 180,E1 -8380.494,E2 -8380.494} C_VEL
LIN {X 0,Y 453.942,Z 970.403,A -85,B 0,C 180,E1 -8381.613,E2 -8381.613} C_VEL
LIN {X 0,Y 454.507,Z 960.596,A -85,B 0,C 180,E1 -8382.65,E2 -8382.65} C_VEL
LIN {X 0,Y 454.972,Z 949.195,A -85,B 0,C 180,E1 -8383.627,E2 -8383.627} C_VEL
LIN {X 0,Y 455.558,Z 937.694,A -85,B 0,C 180,E1 -8384.406,E2 -8384.406} C_VEL
LIN {X 0,Y 455.971,Z 925.896,A -85,B 0,C 180,E1 -8385.02,E2 -8385.02} C_VEL
LIN {X 0,Y 455.656,Z 920.724,A -85,B 0,C 180,E1 -8385.251,E2 -8385.251} C_VEL
LIN {X 0,Y 454.24,Z 908.379,A -85,B 0,C 180,E1 -8385.701,E2 -8385.701} C_VEL
LIN {X 0,Y 453.357,Z 899.174,A -85,B 0,C 180,E1 -8385.946,E2 -8385.946} C_VEL
LIN {X 0,Y 453.724,Z 886.127,A -85,B 0,C 180,E1 -8388.984,E2 -8388.984} C_VEL
LIN {X 0,Y 454.175,Z 870.876,A -85,B 0,C 180,E1 -8392.52,E2 -8392.52} C_VEL
LIN {X 0,Y 454.671,Z 857.442,A -85,B 0,C 180,E1 -8395.647,E2 -8395.647} C_VEL
LIN {X 0,Y 455.132,Z 844.889,A -85,B 0,C 180,E1 -8398.601,E2 -8398.601} C_VEL
LIN {X 0,Y 455.812,Z 829.615,A -85,B 0,C 180,E1 -8402.274,E2 -8402.274} C_VEL
LIN {X 0,Y 456.413,Z 816.709,A -85,B 0,C 180,E1 -8405.501,E2 -8405.501} C_VEL
LIN {X 0,Y 456.394,Z 811.302,A -85,B 0,C 180,E1 -8406.911,E2 -8406.911} C_VEL
LIN {X 0,Y 454.619,Z 801.777,A -85,B 0,C 180,E1 -8409.62,E2 -8409.62} C_VEL
LIN {X 0,Y 453.464,Z 795.998,A -85,B 0,C 180,E1 -8411.348,E2 -8411.348} C_VEL
LIN {X 0,Y 453.461,Z 796.001,A -85,B 0,C 180,E1 -8414.526,E2 -8414.526} C_VEL
LIN {X 0,Y 453.44,Z 796.002,A -85,B 0,C 180,E1 -8418.205,E2 -8418.205} C_VEL
LIN {X 0,Y 453.425,Z 796.002,A -85,B 0,C 180,E1 -8420.806,E2 -8420.806} C_VEL
LIN {X 0,Y 453.409,Z 796.008,A -85,B 0,C 180,E1 -8423.913,E2 -8423.913} C_VEL
LIN {X 0,Y 453.458,Z 795.999,A -85,B 0,C 180,E1 -8427.149,E2 -8427.149} C_VEL
LIN {X 0,Y 453.452,Z 796.003,A -85,B 0,C 180,E1 -8430.267,E2 -8430.267} C_VEL
LIN {X 0,Y 453.415,Z 796.004,A -85,B 0,C 180,E1 -8433.288,E2 -8433.288} C_VEL
LIN {X 0,Y 453.473,Z 796.001,A -85,B 0,C 180,E1 -8436.237,E2 -8436.237} C_VEL
LIN {X 0,Y 453.437,Z 796.002,A -85,B 0,C 180,E1 -8439.115,E2 -8439.115} C_VEL
LIN {X 0,Y 453.444,Z 796.004,A -85,B 0,C 180,E1 -8441.942,E2 -8441.942} C_VEL
LIN {X 0,Y 453.505,Z 795.997,A -85,B 0,C 180,E1 -8445.041,E2 -8445.041} C_VEL
LIN {X 0,Y 456.386,Z 805.992,A -85,B 0,C 180,E1 -8445.736,E2 -8445.736} C_VEL
LIN {X 0,Y 456.082,Z 817.583,A -85,B 0,C 180,E1 -8446.549,E2 -8446.549} C_VEL
LIN {X 0,Y 455.755,Z 826.407,A -85,B 0,C 180,E1 -8447.306,E2 -8447.306} C_VEL
LIN {X 0,Y 455.364,Z 835.071,A -85,B 0,C 180,E1 -8448.2,E2 -8448.2} C_VEL
LIN {X 0,Y 454.914,Z 844.093,A -85,B 0,C 180,E1 -8449.316,E2 -8449.316} C_VEL
LIN {X 0,Y 454.551,Z 851.275,A -85,B 0,C 180,E1 -8450.432,E2 -8450.432} C_VEL
LIN {X 0,Y 454.169,Z 857.339,A -85,B 0,C 180,E1 -8451.546,E2 -8451.546} C_VEL
LIN {X 0,Y 453.976,Z 861.956,A -85,B 0,C 180,E1 -8452.565,E2 -8452.565} C_VEL
LIN {X 0,Y 453.752,Z 866.532,A -85,B 0,C 180,E1 -8453.776,E2 -8453.776} C_VEL
LIN {X 0,Y 453.459,Z 869.277,A -85,B 0,C 180,E1 -8454.664,E2 -8454.664} C_VEL
LIN {X 0,Y 453.289,Z 873.165,A -85,B 0,C 180,E1 -8456.444,E2 -8456.444} C_VEL
LIN {X 0,Y 453.301,Z 874.58,A -85,B 0,C 180,E1 -8457.334,E2 -8457.334} C_VEL
LIN {X 0,Y 453.118,Z 876.021,A -85,B 0,C 180,E1 -8459.111,E2 -8459.111} C_VEL
LIN {X 0,Y 453.108,Z 876.16,A -85,B 0,C 180,E1 -8460,E2 -8460} C_VEL
LIN {X 0,Y 453.068,Z 875.883,A -85,B 0,C 180,E1 -8460.889,E2 -8460.889} C_VEL
LIN {X 0,Y 453.101,Z 874.108,A -85,B 0,C 180,E1 -8462.667,E2 -8462.667} C_VEL
LIN {X 0,Y 453.298,Z 870.652,A -85,B 0,C 180,E1 -8464.446,E2 -8464.446} C_VEL
LIN {X 0,Y 453.444,Z 866.907,A -85,B 0,C 180,E1 -8465.782,E2 -8465.782} C_VEL
LIN {X 0,Y 453.684,Z 862.026,A -85,B 0,C 180,E1 -8467.119,E2 -8467.119} C_VEL
LIN {X 0,Y 453.898,Z 857.036,A -85,B 0,C 180,E1 -8468.235,E2 -8468.235} C_VEL
LIN {X 0,Y 454.258,Z 849.705,A -85,B 0,C 180,E1 -8469.574,E2 -8469.574} C_VEL
LIN {X 0,Y 454.553,Z 842.094,A -85,B 0,C 180,E1 -8470.692,E2 -8470.692} C_VEL
LIN {X 0,Y 454.92,Z 834.963,A -85,B 0,C 180,E1 -8471.586,E2 -8471.586} C_VEL
LIN {X 0,Y 455.22,Z 826.539,A -85,B 0,C 180,E1 -8472.483,E2 -8472.483} C_VEL
LIN {X 0,Y 455.701,Z 816.469,A -85,B 0,C 180,E1 -8473.376,E2 -8473.376} C_VEL
LIN {X 0,Y 456.023,Z 806.745,A -85,B 0,C 180,E1 -8474.061,E2 -8474.061} C_VEL
LIN {X 0,Y 455.504,Z 803.465,A -85,B 0,C 180,E1 -8474.292,E2 -8474.292} C_VEL
LIN {X 0,Y 453.494,Z 795.996,A -85,B 0,C 180,E1 -8474.787,E2 -8474.787} C_VEL
LIN {X 0,Y 453.444,Z 796,A -85,B 0,C 180,E1 -8478.058,E2 -8478.058} C_VEL
LIN {X 0,Y 453.478,Z 795.995,A -85,B 0,C 180,E1 -8481.582,E2 -8481.582} C_VEL
LIN {X 0,Y 453.454,Z 795.996,A -85,B 0,C 180,E1 -8484.738,E2 -8484.738} C_VEL
LIN {X 0,Y 453.463,Z 795.998,A -85,B 0,C 180,E1 -8487.941,E2 -8487.941} C_VEL
LIN {X 0,Y 453.459,Z 795.994,A -85,B 0,C 180,E1 -8490.761,E2 -8490.761} C_VEL
LIN {X 0,Y 453.47,Z 795.998,A -85,B 0,C 180,E1 -8493.913,E2 -8493.913} C_VEL
LIN {X 0,Y 453.44,Z 795.996,A -85,B 0,C 180,E1 -8497.191,E2 -8497.191} C_VEL
LIN {X 0,Y 453.476,Z 795.994,A -85,B 0,C 180,E1 -8500.611,E2 -8500.611} C_VEL
LIN {X 0,Y 453.465,Z 796.001,A -85,B 0,C 180,E1 -8504.221,E2 -8504.221} C_VEL
LIN {X 0,Y 453.454,Z 795.996,A -85,B 0,C 180,E1 -8507.003,E2 -8507.003} C_VEL
LIN {X 0,Y 453.477,Z 795.994,A -85,B 0,C 180,E1 -8509.412,E2 -8509.412} C_VEL
LIN {X 0,Y 453.456,Z 795.995,A -85,B 0,C 180,E1 -8512.809,E2 -8512.809} C_VEL
LIN {X 0,Y 453.474,Z 796,A -85,B 0,C 180,E1 -8516.086,E2 -8516.086} C_VEL
LIN {X 0,Y 453.482,Z 795.991,A -85,B 0,C 180,E1 -8519.24,E2 -8519.24} C_VEL
LIN {X 0,Y 453.539,Z 795.99,A -85,B 0,C 180,E1 -8522.296,E2 -8522.296} C_VEL
LIN {X 0,Y 453.499,Z 795.986,A -85,B 0,C 180,E1 -8525.263,E2 -8525.263} C_VEL
LIN {X 0,Y 453.487,Z 796,A -85,B 0,C 180,E1 -8528.414,E2 -8528.414} C_VEL
LIN {X 0,Y 453.528,Z 795.994,A -85,B 0,C 180,E1 -8531.007,E2 -8531.007} C_VEL
LIN {X 0,Y 453.563,Z 795.987,A -85,B 0,C 180,E1 -8534.026,E2 -8534.026} C_VEL
LIN {X 0,Y 453.525,Z 795.991,A -85,B 0,C 180,E1 -8534.897,E2 -8534.897} C_VEL
LIN {X 0,Y 456.743,Z 807.218,A -85,B 0,C 180,E1 -8535.632,E2 -8535.632} C_VEL
LIN {X 0,Y 456.567,Z 817.711,A -85,B 0,C 180,E1 -8536.353,E2 -8536.353} C_VEL
LIN {X 0,Y 456.473,Z 819.542,A -85,B 0,C 180,E1 -8536.498,E2 -8536.498} C_VEL
LIN {X 0,Y 455.581,Z 824.544,A -85,B 0,C 180,E1 -8536.884,E2 -8536.884} C_VEL
LIN {X 0,Y 452.398,Z 832.485,A -85,B 0,C 180,E1 -8537.518,E2 -8537.518} C_VEL
LIN {X 0,Y 449.233,Z 839.959,A -85,B 0,C 180,E1 -8538.237,E2 -8538.237} C_VEL
LIN {X 0,Y 448.376,Z 844.172,A -85,B 0,C 180,E1 -8538.75,E2 -8538.75} C_VEL
LIN {X 0,Y 447.832,Z 852.926,A -85,B 0,C 180,E1 -8540.058,E2 -8540.058} C_VEL
LIN {X 0,Y 447.364,Z 860.21,A -85,B 0,C 180,E1 -8541.416,E2 -8541.416} C_VEL
LIN {X 0,Y 447.151,Z 866.022,A -85,B 0,C 180,E1 -8542.775,E2 -8542.775} C_VEL
LIN {X 0,Y 446.703,Z 870.653,A -85,B 0,C 180,E1 -8544.129,E2 -8544.129} C_VEL
LIN {X 0,Y 446.496,Z 874.173,A -85,B 0,C 180,E1 -8545.485,E2 -8545.485} C_VEL
LIN {X 0,Y 446.368,Z 875.995,A -85,B 0,C 180,E1 -8546.388,E2 -8546.388} C_VEL
LIN {X 0,Y 446.382,Z 877.353,A -85,B 0,C 180,E1 -8547.291,E2 -8547.291} C_VEL
LIN {X 0,Y 446.238,Z 878.341,A -85,B 0,C 180,E1 -8548.193,E2 -8548.193} C_VEL
LIN {X 0,Y 446.299,Z 879.158,A -85,B 0,C 180,E1 -8549.998,E2 -8549.998} C_VEL
LIN {X 0,Y 446.285,Z 878.98,A -85,B 0,C 180,E1 -8550.901,E2 -8550.901} C_VEL
LIN {X 0,Y 446.238,Z 878.424,A -85,B 0,C 180,E1 -8551.803,E2 -8551.803} C_VEL
LIN {X 0,Y 446.38,Z 877.471,A -85,B 0,C 180,E1 -8552.706,E2 -8552.706} C_VEL
LIN {X 0,Y 446.361,Z 876.165,A -85,B 0,C 180,E1 -8553.609,E2 -8553.609} C_VEL
LIN {X 0,Y 446.549,Z 873.363,A -85,B 0,C 180,E1 -8554.964,E2 -8554.964} C_VEL
LIN {X 0,Y 446.928,Z 869.541,A -85,B 0,C 180,E1 -8556.318,E2 -8556.318} C_VEL
LIN {X 0,Y 447.198,Z 864.398,A -85,B 0,C 180,E1 -8557.737,E2 -8557.737} C_VEL
LIN {X 0,Y 447.541,Z 857.274,A -85,B 0,C 180,E1 -8559.261,E2 -8559.261} C_VEL
LIN {X 0,Y 448.087,Z 849.258,A -85,B 0,C 180,E1 -8560.618,E2 -8560.618} C_VEL
LIN {X 0,Y 448.593,Z 841.04,A -85,B 0,C 180,E1 -8561.75,E2 -8561.75} C_VEL
LIN {X 0,Y 449.068,Z 830.88,A -85,B 0,C 180,E1 -8562.884,E2 -8562.884} C_VEL
LIN {X 0,Y 449.726,Z 820,A -85,B 0,C 180,E1 -8563.849,E2 -8563.849} C_VEL
LIN {X 0,Y 450.013,Z 809.727,A -85,B 0,C 180,E1 -8564.584,E2 -8564.584} C_VEL
LIN {X 0,Y 447.385,Z 800.045,A -85,B 0,C 180,E1 -8565.254,E2 -8565.254} C_VEL
LIN {X 0,Y 446.511,Z 796.868,A -85,B 0,C 180,E1 -8565.46,E2 -8565.46} C_VEL
LIN {X 0,Y 446.457,Z 796.871,A -85,B 0,C 180,E1 -8568.349,E2 -8568.349} C_VEL
LIN {X 0,Y 446.446,Z 796.877,A -85,B 0,C 180,E1 -8571.753,E2 -8571.753} C_VEL
LIN {X 0,Y 446.454,Z 796.87,A -85,B 0,C 180,E1 -8575.15,E2 -8575.15} C_VEL
LIN {X 0,Y 446.48,Z 796.871,A -85,B 0,C 180,E1 -8578.177,E2 -8578.177} C_VEL
LIN {X 0,Y 446.415,Z 796.879,A -85,B 0,C 180,E1 -8581.773,E2 -8581.773} C_VEL
LIN {X 0,Y 446.424,Z 796.876,A -85,B 0,C 180,E1 -8584.521,E2 -8584.521} C_VEL
LIN {X 0,Y 446.428,Z 796.879,A -85,B 0,C 180,E1 -8588.081,E2 -8588.081} C_VEL
LIN {X 0,Y 446.438,Z 796.872,A -85,B 0,C 180,E1 -8590.919,E2 -8590.919} C_VEL
LIN {X 0,Y 446.435,Z 796.873,A -85,B 0,C 180,E1 -8593.839,E2 -8593.839} C_VEL
LIN {X 0,Y 446.436,Z 796.876,A -85,B 0,C 180,E1 -8596.395,E2 -8596.395} C_VEL
LIN {X 0,Y 446.457,Z 796.869,A -85,B 0,C 180,E1 -8599.803,E2 -8599.803} C_VEL
LIN {X 0,Y 446.422,Z 796.872,A -85,B 0,C 180,E1 -8602.122,E2 -8602.122} C_VEL
LIN {X 0,Y 446.417,Z 796.869,A -85,B 0,C 180,E1 -8605.476,E2 -8605.476} C_VEL
LIN {X 0,Y 446.406,Z 796.88,A -85,B 0,C 180,E1 -8608.699,E2 -8608.699} C_VEL
LIN {X 0,Y 446.47,Z 796.866,A -85,B 0,C 180,E1 -8611.82,E2 -8611.82} C_VEL
LIN {X 0,Y 446.443,Z 796.874,A -85,B 0,C 180,E1 -8614.847,E2 -8614.847} C_VEL
LIN {X 0,Y 446.432,Z 796.871,A -85,B 0,C 180,E1 -8618.244,E2 -8618.244} C_VEL
LIN {X 0,Y 446.44,Z 796.871,A -85,B 0,C 180,E1 -8621.648,E2 -8621.648} C_VEL
LIN {X 0,Y 446.491,Z 796.861,A -85,B 0,C 180,E1 -8624.479,E2 -8624.479} C_VEL
LIN {X 0,Y 446.525,Z 796.86,A -85,B 0,C 180,E1 -8628.193,E2 -8628.193} C_VEL
LIN {X 0,Y 446.583,Z 796.854,A -85,B 0,C 180,E1 -8631.857,E2 -8631.857} C_VEL
LIN {X 0,Y 446.624,Z 796.85,A -85,B 0,C 180,E1 -8634.582,E2 -8634.582} C_VEL
LIN {X 0,Y 446.691,Z 796.843,A -85,B 0,C 180,E1 -8637.295,E2 -8637.295} C_VEL
LIN {X 0,Y 446.774,Z 796.833,A -85,B 0,C 180,E1 -8640,E2 -8640} C_VEL
LIN {X 0,Y 446.674,Z 796.843,A -85,B 0,C 180,E1 -8642.705,E2 -8642.705} C_VEL
LIN {X 0,Y 446.6,Z 796.851,A -85,B 0,C 180,E1 -8646.324,E2 -8646.324} C_VEL
LIN {X 0,Y 446.52,Z 796.861,A -85,B 0,C 180,E1 -8649.056,E2 -8649.056} C_VEL
LIN {X 0,Y 446.516,Z 796.858,A -85,B 0,C 180,E1 -8652.73,E2 -8652.73} C_VEL
LIN {X 0,Y 446.471,Z 796.869,A -85,B 0,C 180,E1 -8656.46,E2 -8656.46} C_VEL
LIN {X 0,Y 446.451,Z 796.871,A -85,B 0,C 180,E1 -8659.304,E2 -8659.304} C_VEL
LIN {X 0,Y 446.401,Z 796.882,A -85,B 0,C 180,E1 -8662.201,E2 -8662.201} C_VEL
LIN {X 0,Y 446.422,Z 796.872,A -85,B 0,C 180,E1 -8665.155,E2 -8665.155} C_VEL
LIN {X 0,Y 446.424,Z 796.878,A -85,B 0,C 180,E1 -8668.183,E2 -8668.183} C_VEL
LIN {X 0,Y 446.4,Z 796.876,A -85,B 0,C 180,E1 -8671.302,E2 -8671.302} C_VEL
LIN {X 0,Y 446.407,Z 796.88,A -85,B 0,C 180,E1 -8674.525,E2 -8674.525} C_VEL
LIN {X 0,Y 446.385,Z 796.883,A -85,B 0,C 180,E1 -8678.078,E2 -8678.078} C_VEL
LIN {X 0,Y 446.389,Z 796.878,A -85,B 0,C 180,E1 -8681.396,E2 -8681.396} C_VEL
LIN {X 0,Y 446.407,Z 796.878,A -85,B 0,C 180,E1 -8684.894,E2 -8684.894} C_VEL
LIN {X 0,Y 446.434,Z 796.975,A -85,B 0,C 180,E1 -8688.36,E2 -8688.36} C_VEL
LIN {X 0,Y 448.551,Z 807.679,A -85,B 0,C 180,E1 -8691.574,E2 -8691.574} C_VEL
LIN {X 0,Y 449.564,Z 813.531,A -85,B 0,C 180,E1 -8693.232,E2 -8693.232} C_VEL
LIN {X 0,Y 449.196,Z 823.099,A -85,B 0,C 180,E1 -8695.722,E2 -8695.722} C_VEL
LIN {X 0,Y 448.582,Z 835.672,A -85,B 0,C 180,E1 -8698.87,E2 -8698.87} C_VEL
LIN {X 0,Y 447.921,Z 850.322,A -85,B 0,C 180,E1 -8702.43,E2 -8702.43} C_VEL
LIN {X 0,Y 447.408,Z 863.828,A -85,B 0,C 180,E1 -8705.655,E2 -8705.655} C_VEL
LIN {X 0,Y 446.868,Z 878.112,A -85,B 0,C 180,E1 -8709.037,E2 -8709.037} C_VEL
LIN {X 0,Y 446.53,Z 891.16,A -85,B 0,C 180,E1 -8712.129,E2 -8712.129} C_VEL
LIN {X 0,Y 446.301,Z 898.212,A -85,B 0,C 180,E1 -8713.809,E2 -8713.809} C_VEL
LIN {X 0,Y 447.695,Z 912.689,A -85,B 0,C 180,E1 -8714.223,E2 -8714.223} C_VEL
LIN {X 0,Y 449.098,Z 924.915,A -85,B 0,C 180,E1 -8714.748,E2 -8714.748} C_VEL
LIN {X 0,Y 448.613,Z 936.689,A -85,B 0,C 180,E1 -8715.37,E2 -8715.37} C_VEL
LIN {X 0,Y 447.979,Z 948.182,A -85,B 0,C 180,E1 -8716.16,E2 -8716.16} C_VEL
LIN {X 0,Y 447.416,Z 959.517,A -85,B 0,C 180,E1 -8717.146,E2 -8717.146} C_VEL
LIN {X 0,Y 446.856,Z 969.368,A -85,B 0,C 180,E1 -8718.204,E2 -8718.204} C_VEL
LIN {X 0,Y 446.431,Z 978.031,A -85,B 0,C 180,E1 -8719.342,E2 -8719.342} C_VEL
LIN {X 0,Y 446.1,Z 986.509,A -85,B 0,C 180,E1 -8720.709,E2 -8720.709} C_VEL
LIN {X 0,Y 445.864,Z 993.36,A -85,B 0,C 180,E1 -8722.074,E2 -8722.074} C_VEL
LIN {X 0,Y 445.744,Z 999.654,A -85,B 0,C 180,E1 -8723.665,E2 -8723.665} C_VEL
LIN {X 0,Y 445.711,Z 1003.756,A -85,B 0,C 180,E1 -8725.027,E2 -8725.027} C_VEL
LIN {X 0,Y 445.724,Z 1006.793,A -85,B 0,C 180,E1 -8726.386,E2 -8726.386} C_VEL
LIN {X 0,Y 445.665,Z 1008.229,A -85,B 0,C 180,E1 -8727.29,E2 -8727.29} C_VEL
LIN {X 0,Y 445.664,Z 1009.258,A -85,B 0,C 180,E1 -8728.194,E2 -8728.194} C_VEL
LIN {X 0,Y 445.642,Z 1009.883,A -85,B 0,C 180,E1 -8729.098,E2 -8729.098} C_VEL
LIN {X 0,Y 445.637,Z 1010.104,A -85,B 0,C 180,E1 -8730.002,E2 -8730.002} C_VEL
LIN {X 0,Y 445.642,Z 1009.881,A -85,B 0,C 180,E1 -8730.905,E2 -8730.905} C_VEL
LIN {X 0,Y 445.664,Z 1009.254,A -85,B 0,C 180,E1 -8731.809,E2 -8731.809} C_VEL
LIN {X 0,Y 445.665,Z 1008.222,A -85,B 0,C 180,E1 -8732.713,E2 -8732.713} C_VEL
LIN {X 0,Y 445.725,Z 1006.784,A -85,B 0,C 180,E1 -8733.618,E2 -8733.618} C_VEL
LIN {X 0,Y 445.712,Z 1003.748,A -85,B 0,C 180,E1 -8734.977,E2 -8734.977} C_VEL
LIN {X 0,Y 445.71,Z 998.743,A -85,B 0,C 180,E1 -8736.589,E2 -8736.589} C_VEL
LIN {X 0,Y 445.902,Z 992.308,A -85,B 0,C 180,E1 -8738.157,E2 -8738.157} C_VEL
LIN {X 0,Y 446.166,Z 985.228,A -85,B 0,C 180,E1 -8739.522,E2 -8739.522} C_VEL
LIN {X 0,Y 446.548,Z 976.39,A -85,B 0,C 180,E1 -8740.888,E2 -8740.888} C_VEL
LIN {X 0,Y 446.983,Z 967.359,A -85,B 0,C 180,E1 -8742.026,E2 -8742.026} C_VEL
LIN {X 0,Y 447.608,Z 957.298,A -85,B 0,C 180,E1 -8743.065,E2 -8743.065} C_VEL
LIN {X 0,Y 448.037,Z 946.688,A -85,B 0,C 180,E1 -8743.957,E2 -8743.957} C_VEL
LIN {X 0,Y 448.72,Z 934.693,A -85,B 0,C 180,E1 -8744.746,E2 -8744.746} C_VEL
LIN {X 0,Y 448.985,Z 923.514,A -85,B 0,C 180,E1 -8745.318,E2 -8745.318} C_VEL
LIN {X 0,Y 447.587,Z 911.323,A -85,B 0,C 180,E1 -8745.823,E2 -8745.823} C_VEL
LIN {X 0,Y 446.283,Z 898.189,A -85,B 0,C 180,E1 -8746.2,E2 -8746.2} C_VEL
LIN {X 0,Y 446.681,Z 885.173,A -85,B 0,C 180,E1 -8749.295,E2 -8749.295} C_VEL
LIN {X 0,Y 447.174,Z 869.953,A -85,B 0,C 180,E1 -8752.893,E2 -8752.893} C_VEL
LIN {X 0,Y 447.685,Z 856.549,A -85,B 0,C 180,E1 -8756.077,E2 -8756.077} C_VEL
LIN {X 0,Y 448.203,Z 842.974,A -85,B 0,C 180,E1 -8759.343,E2 -8759.343} C_VEL
LIN {X 0,Y 448.799,Z 831.071,A -85,B 0,C 180,E1 -8762.262,E2 -8762.262} C_VEL
LIN {X 0,Y 449.41,Z 818.891,A -85,B 0,C 180,E1 -8765.355,E2 -8765.355} C_VEL
LIN {X 0,Y 449.517,Z 813.514,A -85,B 0,C 180,E1 -8766.771,E2 -8766.771} C_VEL
LIN {X 0,Y 447.979,Z 804.747,A -85,B 0,C 180,E1 -8769.276,E2 -8769.276} C_VEL
LIN {X 0,Y 446.417,Z 796.876,A -85,B 0,C 180,E1 -8771.695,E2 -8771.695} C_VEL
LIN {X 0,Y 446.402,Z 796.883,A -85,B 0,C 180,E1 -8775.112,E2 -8775.112} C_VEL
LIN {X 0,Y 446.399,Z 796.878,A -85,B 0,C 180,E1 -8778.605,E2 -8778.605} C_VEL
LIN {X 0,Y 446.386,Z 796.882,A -85,B 0,C 180,E1 -8782.119,E2 -8782.119} C_VEL
LIN {X 0,Y 446.385,Z 796.882,A -85,B 0,C 180,E1 -8785.473,E2 -8785.473} C_VEL
LIN {X 0,Y 446.393,Z 796.879,A -85,B 0,C 180,E1 -8788.698,E2 -8788.698} C_VEL
LIN {X 0,Y 446.402,Z 796.88,A -85,B 0,C 180,E1 -8791.843,E2 -8791.843} C_VEL
LIN {X 0,Y 446.404,Z 796.877,A -85,B 0,C 180,E1 -8794.844,E2 -8794.844} C_VEL
LIN {X 0,Y 446.446,Z 796.878,A -85,B 0,C 180,E1 -8798.248,E2 -8798.248} C_VEL
LIN {X 0,Y 446.398,Z 796.88,A -85,B 0,C 180,E1 -8801.647,E2 -8801.647} C_VEL
LIN {X 0,Y 446.446,Z 796.877,A -85,B 0,C 180,E1 -8804.77,E2 -8804.77} C_VEL
LIN {X 0,Y 449.607,Z 807.458,A -85,B 0,C 180,E1 -8805.516,E2 -8805.516} C_VEL
LIN {X 0,Y 449.307,Z 818.918,A -85,B 0,C 180,E1 -8806.339,E2 -8806.339} C_VEL
LIN {X 0,Y 448.945,Z 827.734,A -85,B 0,C 180,E1 -8807.11,E2 -8807.11} C_VEL
LIN {X 0,Y 448.527,Z 836.357,A -85,B 0,C 180,E1 -8808.017,E2 -8808.017} C_VEL
LIN {X 0,Y 448.075,Z 845.344,A -85,B 0,C 180,E1 -8809.151,E2 -8809.151} C_VEL
LIN {X 0,Y 447.664,Z 852.503,A -85,B 0,C 180,E1 -8810.284,E2 -8810.284} C_VEL
LIN {X 0,Y 447.265,Z 858.548,A -85,B 0,C 180,E1 -8811.415,E2 -8811.415} C_VEL
LIN {X 0,Y 447.07,Z 862.993,A -85,B 0,C 180,E1 -8812.41,E2 -8812.41} C_VEL
LIN {X 0,Y 446.792,Z 867.709,A -85,B 0,C 180,E1 -8813.678,E2 -8813.678} C_VEL
LIN {X 0,Y 446.487,Z 870.442,A -85,B 0,C 180,E1 -8814.581,E2 -8814.581} C_VEL
LIN {X 0,Y 446.321,Z 874.299,A -85,B 0,C 180,E1 -8816.389,E2 -8816.389} C_VEL
LIN {X 0,Y 446.323,Z 875.701,A -85,B 0,C 180,E1 -8817.292,E2 -8817.292} C_VEL
LIN {X 0,Y 446.123,Z 877.116,A -85,B 0,C 180,E1 -8819.097,E2 -8819.097} C_VEL
LIN {X 0,Y 446.108,Z 877.239,A -85,B 0,C 180,E1 -8820,E2 -8820} C_VEL
LIN {X 0,Y 446.077,Z 876.939,A -85,B 0,C 180,E1 -8820.903,E2 -8820.903} C_VEL
LIN {X 0,Y 446.084,Z 875.134,A -85,B 0,C 180,E1 -8822.709,E2 -8822.709} C_VEL
LIN {X 0,Y 446.287,Z 871.623,A -85,B 0,C 180,E1 -8824.516,E2 -8824.516} C_VEL
LIN {X 0,Y 446.452,Z 867.836,A -85,B 0,C 180,E1 -8825.873,E2 -8825.873} C_VEL
LIN {X 0,Y 446.71,Z 862.909,A -85,B 0,C 180,E1 -8827.231,E2 -8827.231} C_VEL
LIN {X 0,Y 446.943,Z 857.873,A -85,B 0,C 180,E1 -8828.364,E2 -8828.364} C_VEL
LIN {X 0,Y 447.324,Z 850.492,A -85,B 0,C 180,E1 -8829.724,E2 -8829.724} C_VEL
LIN {X 0,Y 447.612,Z 842.82,A -85,B 0,C 180,E1 -8830.86,E2 -8830.86} C_VEL
LIN {X 0,Y 447.995,Z 835.63,A -85,B 0,C 180,E1 -8831.768,E2 -8831.768} C_VEL
LIN {X 0,Y 448.337,Z 827.134,A -85,B 0,C 180,E1 -8832.677,E2 -8832.677} C_VEL
LIN {X 0,Y 448.825,Z 817.002,A -85,B 0,C 180,E1 -8833.585,E2 -8833.585} C_VEL
LIN {X 0,Y 449.119,Z 807.019,A -85,B 0,C 180,E1 -8834.291,E2 -8834.291} C_VEL
LIN {X 0,Y 446.949,Z 798.818,A -85,B 0,C 180,E1 -8834.866,E2 -8834.866} C_VEL
LIN {X 0,Y 446.447,Z 796.875,A -85,B 0,C 180,E1 -8834.997,E2 -8834.997} C_VEL
LIN {X 0,Y 446.384,Z 796.884,A -85,B 0,C 180,E1 -8837.406,E2 -8837.406} C_VEL
LIN {X 0,Y 446.388,Z 796.874,A -85,B 0,C 180,E1 -8840.266,E2 -8840.266} C_VEL
LIN {X 0,Y 446.407,Z 796.874,A -85,B 0,C 180,E1 -8843.178,E2 -8843.178} C_VEL
LIN {X 0,Y 446.422,Z 796.87,A -85,B 0,C 180,E1 -8846.186,E2 -8846.186} C_VEL
LIN {X 0,Y 446.421,Z 796.871,A -85,B 0,C 180,E1 -8849.212,E2 -8849.212} C_VEL
LIN {X 0,Y 446.421,Z 796.868,A -85,B 0,C 180,E1 -8852.362,E2 -8852.362} C_VEL
LIN {X 0,Y 446.415,Z 796.876,A -85,B 0,C 180,E1 -8855.627,E2 -8855.627} C_VEL
LIN {X 0,Y 446.404,Z 796.873,A -85,B 0,C 180,E1 -8859.031,E2 -8859.031} C_VEL
LIN {X 0,Y 446.39,Z 796.879,A -85,B 0,C 180,E1 -8862.27,E2 -8862.27} C_VEL
LIN {X 0,Y 446.456,Z 796.868,A -85,B 0,C 180,E1 -8865.103,E2 -8865.103} C_VEL
LIN {X 0,Y 446.417,Z 796.875,A -85,B 0,C 180,E1 -8868.606,E2 -8868.606} C_VEL
LIN {X 0,Y 446.417,Z 796.879,A -85,B 0,C 180,E1 -8871.921,E2 -8871.921} C_VEL
LIN {X 0,Y 446.429,Z 796.872,A -85,B 0,C 180,E1 -8875.476,E2 -8875.476} C_VEL
LIN {X 0,Y 446.422,Z 796.873,A -85,B 0,C 180,E1 -8878.699,E2 -8878.699} C_VEL
LIN {X 0,Y 446.492,Z 796.863,A -85,B 0,C 180,E1 -8881.82,E2 -8881.82} C_VEL
LIN {X 0,Y 446.443,Z 796.867,A -85,B 0,C 180,E1 -8884.845,E2 -8884.845} C_VEL
LIN {X 0,Y 446.455,Z 796.874,A -85,B 0,C 180,E1 -8888.244,E2 -8888.244} C_VEL
LIN {X 0,Y 446.457,Z 796.874,A -85,B 0,C 180,E1 -8891.648,E2 -8891.648} C_VEL
LIN {X 0,Y 446.517,Z 796.999,A -85,B 0,C 180,E1 -8894.654,E2 -8894.654} C_VEL
LIN {X 0,Y 449.826,Z 808.274,A -85,B 0,C 180,E1 -8895.407,E2 -8895.407} C_VEL
LIN {X 0,Y 449.76,Z 818.74,A -85,B 0,C 180,E1 -8896.142,E2 -8896.142} C_VEL
LIN {X 0,Y 449.208,Z 828.755,A -85,B 0,C 180,E1 -8897.001,E2 -8897.001} C_VEL
LIN {X 0,Y 448.703,Z 838.354,A -85,B 0,C 180,E1 -8898.021,E2 -8898.021} C_VEL
LIN {X 0,Y 448.376,Z 844.172,A -85,B 0,C 180,E1 -8898.75,E2 -8898.75} C_VEL
LIN {X 0,Y 447.535,Z 848.233,A -85,B 0,C 180,E1 -8899.291,E2 -8899.291} C_VEL
LIN {X 0,Y 444.405,Z 854.614,A -85,B 0,C 180,E1 -8900.177,E2 -8900.177} C_VEL
LIN {X 0,Y 441.23,Z 860.406,A -85,B 0,C 180,E1 -8901.133,E2 -8901.133} C_VEL
LIN {X 0,Y 440.332,Z 863.491,A -85,B 0,C 180,E1 -8901.776,E2 -8901.776} C_VEL
LIN {X 0,Y 440.078,Z 868.718,A -85,B 0,C 180,E1 -8903.119,E2 -8903.119} C_VEL
LIN {X 0,Y 439.585,Z 872.98,A -85,B 0,C 180,E1 -8904.494,E2 -8904.494} C_VEL
LIN {X 0,Y 439.493,Z 875.205,A -85,B 0,C 180,E1 -8905.412,E2 -8905.412} C_VEL
LIN {X 0,Y 439.358,Z 877.027,A -85,B 0,C 180,E1 -8906.33,E2 -8906.33} C_VEL
LIN {X 0,Y 439.369,Z 878.385,A -85,B 0,C 180,E1 -8907.248,E2 -8907.248} C_VEL
LIN {X 0,Y 439.22,Z 879.372,A -85,B 0,C 180,E1 -8908.164,E2 -8908.164} C_VEL
LIN {X 0,Y 439.282,Z 880.188,A -85,B 0,C 180,E1 -8909.998,E2 -8909.998} C_VEL
LIN {X 0,Y 439.271,Z 880.01,A -85,B 0,C 180,E1 -8910.915,E2 -8910.915} C_VEL
LIN {X 0,Y 439.22,Z 879.455,A -85,B 0,C 180,E1 -8911.832,E2 -8911.832} C_VEL
LIN {X 0,Y 439.366,Z 878.502,A -85,B 0,C 180,E1 -8912.749,E2 -8912.749} C_VEL
LIN {X 0,Y 439.351,Z 877.195,A -85,B 0,C 180,E1 -8913.667,E2 -8913.667} C_VEL
LIN {X 0,Y 439.55,Z 874.393,A -85,B 0,C 180,E1 -8915.043,E2 -8915.043} C_VEL
LIN {X 0,Y 439.955,Z 870.57,A -85,B 0,C 180,E1 -8916.419,E2 -8916.419} C_VEL
LIN {X 0,Y 440.25,Z 865.371,A -85,B 0,C 180,E1 -8917.874,E2 -8917.874} C_VEL
LIN {X 0,Y 440.61,Z 858.303,A -85,B 0,C 180,E1 -8919.408,E2 -8919.408} C_VEL
LIN {X 0,Y 441.186,Z 850.286,A -85,B 0,C 180,E1 -8920.786,E2 -8920.786} C_VEL
LIN {X 0,Y 441.718,Z 842.068,A -85,B 0,C 180,E1 -8921.935,E2 -8921.935} C_VEL
LIN {X 0,Y 442.223,Z 831.907,A -85,B 0,C 180,E1 -8923.087,E2 -8923.087} C_VEL
LIN {X 0,Y 442.907,Z 821.019,A -85,B 0,C 180,E1 -8924.067,E2 -8924.067} C_VEL
LIN {X 0,Y 443.178,Z 810.758,A -85,B 0,C 180,E1 -8924.814,E2 -8924.814} C_VEL
LIN {X 0,Y 440.008,Z 799.686,A -85,B 0,C 180,E1 -8925.593,E2 -8925.593} C_VEL
LIN {X 0,Y 439.467,Z 797.746,A -85,B 0,C 180,E1 -8925.714,E2 -8925.714} C_VEL
LIN {X 0,Y 439.44,Z 797.746,A -85,B 0,C 180,E1 -8929.335,E2 -8929.335} C_VEL
LIN {X 0,Y 439.363,Z 797.752,A -85,B 0,C 180,E1 -8932.573,E2 -8932.573} C_VEL
LIN {X 0,Y 439.402,Z 797.752,A -85,B 0,C 180,E1 -8935.583,E2 -8935.583} C_VEL
LIN {X 0,Y 439.413,Z 797.747,A -85,B 0,C 180,E1 -8938.671,E2 -8938.671} C_VEL
LIN {X 0,Y 439.366,Z 797.759,A -85,B 0,C 180,E1 -8942.029,E2 -8942.029} C_VEL
LIN {X 0,Y 439.389,Z 797.75,A -85,B 0,C 180,E1 -8945.339,E2 -8945.339} C_VEL
LIN {X 0,Y 439.387,Z 797.753,A -85,B 0,C 180,E1 -8948.592,E2 -8948.592} C_VEL
LIN {X 0,Y 439.396,Z 797.748,A -85,B 0,C 180,E1 -8951.257,E2 -8951.257} C_VEL
LIN {X 0,Y 439.4,Z 797.751,A -85,B 0,C 180,E1 -8954.726,E2 -8954.726} C_VEL
LIN {X 0,Y 439.401,Z 797.745,A -85,B 0,C 180,E1 -8957.796,E2 -8957.796} C_VEL
LIN {X 0,Y 439.44,Z 797.747,A -85,B 0,C 180,E1 -8960.229,E2 -8960.229} C_VEL
LIN {X 0,Y 439.364,Z 797.752,A -85,B 0,C 180,E1 -8963.712,E2 -8963.712} C_VEL
LIN {X 0,Y 439.359,Z 797.755,A -85,B 0,C 180,E1 -8967.053,E2 -8967.053} C_VEL
LIN {X 0,Y 439.382,Z 797.749,A -85,B 0,C 180,E1 -8970.274,E2 -8970.274} C_VEL
LIN {X 0,Y 439.418,Z 797.743,A -85,B 0,C 180,E1 -8973.587,E2 -8973.587} C_VEL
LIN {X 0,Y 439.371,Z 797.752,A -85,B 0,C 180,E1 -8976.429,E2 -8976.429} C_VEL
LIN {X 0,Y 439.372,Z 797.751,A -85,B 0,C 180,E1 -8979.396,E2 -8979.396} C_VEL
LIN {X 0,Y 439.414,Z 797.746,A -85,B 0,C 180,E1 -8982.309,E2 -8982.309} C_VEL
LIN {X 0,Y 439.43,Z 797.745,A -85,B 0,C 180,E1 -8985.173,E2 -8985.173} C_VEL
LIN {X 0,Y 439.493,Z 797.737,A -85,B 0,C 180,E1 -8988.001,E2 -8988.001} C_VEL
LIN {X 0,Y 439.531,Z 797.734,A -85,B 0,C 180,E1 -8991.726,E2 -8991.726} C_VEL
LIN {X 0,Y 439.599,Z 797.725,A -85,B 0,C 180,E1 -8994.495,E2 -8994.495} C_VEL
LIN {X 0,Y 439.617,Z 797.722,A -85,B 0,C 180,E1 -8998.168,E2 -8998.168} C_VEL
LIN {X 0,Y 439.744,Z 797.708,A -85,B 0,C 180,E1 -9000,E2 -9000} C_VEL
LIN {X 0,Y 439.623,Z 797.722,A -85,B 0,C 180,E1 -9002.749,E2 -9002.749} C_VEL
LIN {X 0,Y 439.572,Z 797.726,A -85,B 0,C 180,E1 -9006.426,E2 -9006.426} C_VEL
LIN {X 0,Y 439.482,Z 797.739,A -85,B 0,C 180,E1 -9009.202,E2 -9009.202} C_VEL
LIN {X 0,Y 439.487,Z 797.733,A -85,B 0,C 180,E1 -9012.727,E2 -9012.727} C_VEL
LIN {X 0,Y 439.428,Z 797.747,A -85,B 0,C 180,E1 -9016.349,E2 -9016.349} C_VEL
LIN {X 0,Y 439.385,Z 797.754,A -85,B 0,C 180,E1 -9019.627,E2 -9019.627} C_VEL
LIN {X 0,Y 439.346,Z 797.757,A -85,B 0,C 180,E1 -9022.576,E2 -9022.576} C_VEL
LIN {X 0,Y 439.36,Z 797.754,A -85,B 0,C 180,E1 -9025.588,E2 -9025.588} C_VEL
LIN {X 0,Y 439.381,Z 797.753,A -85,B 0,C 180,E1 -9028.676,E2 -9028.676} C_VEL
LIN {X 0,Y 439.353,Z 797.759,A -85,B 0,C 180,E1 -9032.031,E2 -9032.031} C_VEL
LIN {X 0,Y 439.374,Z 797.752,A -85,B 0,C 180,E1 -9035.341,E2 -9035.341} C_VEL
LIN {X 0,Y 439.341,Z 797.761,A -85,B 0,C 180,E1 -9038.599,E2 -9038.599} C_VEL
LIN {X 0,Y 439.338,Z 797.756,A -85,B 0,C 180,E1 -9042.211,E2 -9042.211} C_VEL
LIN {X 0,Y 439.36,Z 797.758,A -85,B 0,C 180,E1 -9045.269,E2 -9045.269} C_VEL
LIN {X 0,Y 439.381,Z 797.936,A -85,B 0,C 180,E1 -9048.062,E2 -9048.062} C_VEL
LIN {X 0,Y 441.224,Z 807.135,A -85,B 0,C 180,E1 -9050.894,E2 -9050.894} C_VEL
LIN {X 0,Y 442.656,Z 815.007,A -85,B 0,C 180,E1 -9053.179,E2 -9053.179} C_VEL
LIN {X 0,Y 442.207,Z 824.671,A -85,B 0,C 180,E1 -9055.735,E2 -9055.735} C_VEL
LIN {X 0,Y 441.575,Z 836.916,A -85,B 0,C 180,E1 -9058.854,E2 -9058.854} C_VEL
LIN {X 0,Y 440.879,Z 851.519,A -85,B 0,C 180,E1 -9062.468,E2 -9062.468} C_VEL
LIN {X 0,Y 440.334,Z 864.945,A -85,B 0,C 180,E1 -9065.735,E2 -9065.735} C_VEL
LIN {X 0,Y 439.75,Z 880.191,A -85,B 0,C 180,E1 -9069.417,E2 -9069.417} C_VEL
LIN {X 0,Y 439.317,Z 894.108,A -85,B 0,C 180,E1 -9072.787,E2 -9072.787} C_VEL
LIN {X 0,Y 439.247,Z 897.239,A -85,B 0,C 180,E1 -9073.547,E2 -9073.547} C_VEL
LIN {X 0,Y 440.581,Z 911.072,A -85,B 0,C 180,E1 -9073.945,E2 -9073.945} C_VEL
LIN {X 0,Y 441.955,Z 923.831,A -85,B 0,C 180,E1 -9074.495,E2 -9074.495} C_VEL
LIN {X 0,Y 441.807,Z 933.699,A -85,B 0,C 180,E1 -9075.021,E2 -9075.021} C_VEL
LIN {X 0,Y 441.094,Z 945.683,A -85,B 0,C 180,E1 -9075.822,E2 -9075.822} C_VEL
LIN {X 0,Y 440.516,Z 956.888,A -85,B 0,C 180,E1 -9076.786,E2 -9076.786} C_VEL
LIN {X 0,Y 440.003,Z 966.338,A -85,B 0,C 180,E1 -9077.784,E2 -9077.784} C_VEL
LIN {X 0,Y 439.491,Z 975.357,A -85,B 0,C 180,E1 -9078.938,E2 -9078.938} C_VEL
LIN {X 0,Y 439.101,Z 984.193,A -85,B 0,C 180,E1 -9080.327,E2 -9080.327} C_VEL
LIN {X 0,Y 438.86,Z 991.277,A -85,B 0,C 180,E1 -9081.715,E2 -9081.715} C_VEL
LIN {X 0,Y 438.684,Z 997.884,A -85,B 0,C 180,E1 -9083.355,E2 -9083.355} C_VEL
LIN {X 0,Y 438.671,Z 1002.718,A -85,B 0,C 180,E1 -9084.946,E2 -9084.946} C_VEL
LIN {X 0,Y 438.688,Z 1005.758,A -85,B 0,C 180,E1 -9086.328,E2 -9086.328} C_VEL
LIN {X 0,Y 438.629,Z 1007.195,A -85,B 0,C 180,E1 -9087.247,E2 -9087.247} C_VEL
LIN {X 0,Y 438.631,Z 1008.225,A -85,B 0,C 180,E1 -9088.165,E2 -9088.165} C_VEL
LIN {X 0,Y 438.615,Z 1008.851,A -85,B 0,C 180,E1 -9089.084,E2 -9089.084} C_VEL
LIN {X 0,Y 438.613,Z 1009.073,A -85,B 0,C 180,E1 -9090.002,E2 -9090.002} C_VEL
LIN {X 0,Y 438.615,Z 1008.849,A -85,B 0,C 180,E1 -9090.92,E2 -9090.92} C_VEL
LIN {X 0,Y 438.631,Z 1008.221,A -85,B 0,C 180,E1 -9091.838,E2 -9091.838} C_VEL
LIN {X 0,Y 438.63,Z 1007.188,A -85,B 0,C 180,E1 -9092.757,E2 -9092.757} C_VEL
LIN {X 0,Y 438.689,Z 1005.749,A -85,B 0,C 180,E1 -9093.676,E2 -9093.676} C_VEL
LIN {X 0,Y 438.673,Z 1002.71,A -85,B 0,C 180,E1 -9095.057,E2 -9095.057} C_VEL
LIN {X 0,Y 438.646,Z 998.039,A -85,B 0,C 180,E1 -9096.602,E2 -9096.602} C_VEL
LIN {X 0,Y 438.819,Z 992.301,A -85,B 0,C 180,E1 -9098.057,E2 -9098.057} C_VEL
LIN {X 0,Y 439.072,Z 985.446,A -85,B 0,C 180,E1 -9099.445,E2 -9099.445} C_VEL
LIN {X 0,Y 439.417,Z 976.962,A -85,B 0,C 180,E1 -9100.833,E2 -9100.833} C_VEL
LIN {X 0,Y 439.855,Z 968.29,A -85,B 0,C 180,E1 -9101.99,E2 -9101.99} C_VEL
LIN {X 0,Y 440.485,Z 958.679,A -85,B 0,C 180,E1 -9103.04,E2 -9103.04} C_VEL
LIN {X 0,Y 441.008,Z 947.082,A -85,B 0,C 180,E1 -9104.067,E2 -9104.067} C_VEL
LIN {X 0,Y 441.711,Z 935.591,A -85,B 0,C 180,E1 -9104.868,E2 -9104.868} C_VEL
LIN {X 0,Y 441.953,Z 923.758,A -85,B 0,C 180,E1 -9105.508,E2 -9105.508} C_VEL
LIN {X 0,Y 440.697,Z 911.995,A -85,B 0,C 180,E1 -9106.022,E2 -9106.022} C_VEL
LIN {X 0,Y 439.269,Z 898.136,A -85,B 0,C 180,E1 -9106.434,E2 -9106.434} C_VEL
LIN {X 0,Y 439.218,Z 897.146,A -85,B 0,C 180,E1 -9106.471,E2 -9106.471} C_VEL
LIN {X 0,Y 439.612,Z 884.197,A -85,B 0,C 180,E1 -9109.618,E2 -9109.618} C_VEL
LIN {X 0,Y 440.172,Z 869.029,A -85,B 0,C 180,E1 -9113.278,E2 -9113.278} C_VEL
LIN {X 0,Y 440.797,Z 854.634,A -85,B 0,C 180,E1 -9116.765,E2 -9116.765} C_VEL
LIN {X 0,Y 441.313,Z 841.052,A -85,B 0,C 180,E1 -9120.11,E2 -9120.11} C_VEL
LIN {X 0,Y 441.927,Z 829.539,A -85,B 0,C 180,E1 -9123.004,E2 -9123.004} C_VEL
LIN {X 0,Y 442.586,Z 818.091,A -85,B 0,C 180,E1 -9125.984,E2 -9125.984} C_VEL
LIN {X 0,Y 442.491,Z 813.899,A -85,B 0,C 180,E1 -9127.126,E2 -9127.126} C_VEL
LIN {X 0,Y 440.63,Z 804.003,A -85,B 0,C 180,E1 -9130.04,E2 -9130.04} C_VEL
LIN {X 0,Y 439.37,Z 797.755,A -85,B 0,C 180,E1 -9132.018,E2 -9132.018} C_VEL
LIN {X 0,Y 439.357,Z 797.76,A -85,B 0,C 180,E1 -9135.265,E2 -9135.265} C_VEL
LIN {X 0,Y 439.362,Z 797.755,A -85,B 0,C 180,E1 -9138.749,E2 -9138.749} C_VEL
LIN {X 0,Y 439.352,Z 797.757,A -85,B 0,C 180,E1 -9141.613,E2 -9141.613} C_VEL
LIN {X 0,Y 439.35,Z 797.756,A -85,B 0,C 180,E1 -9144.839,E2 -9144.839} C_VEL
LIN {X 0,Y 439.35,Z 797.76,A -85,B 0,C 180,E1 -9148.138,E2 -9148.138} C_VEL
LIN {X 0,Y 439.381,Z 797.753,A -85,B 0,C 180,E1 -9151.324,E2 -9151.324} C_VEL
LIN {X 0,Y 439.344,Z 797.76,A -85,B 0,C 180,E1 -9154.411,E2 -9154.411} C_VEL
LIN {X 0,Y 439.352,Z 797.755,A -85,B 0,C 180,E1 -9157.424,E2 -9157.424} C_VEL
LIN {X 0,Y 439.36,Z 797.76,A -85,B 0,C 180,E1 -9160.372,E2 -9160.372} C_VEL
LIN {X 0,Y 439.4,Z 797.752,A -85,B 0,C 180,E1 -9163.676,E2 -9163.676} C_VEL
LIN {X 0,Y 439.405,Z 797.754,A -85,B 0,C 180,E1 -9164.46,E2 -9164.46} C_VEL
LIN {X 0,Y 442.84,Z 809.036,A -85,B 0,C 180,E1 -9165.29,E2 -9165.29} C_VEL
LIN {X 0,Y 442.531,Z 820.287,A -85,B 0,C 180,E1 -9166.118,E2 -9166.118} C_VEL
LIN {X 0,Y 442.178,Z 829.128,A -85,B 0,C 180,E1 -9166.909,E2 -9166.909} C_VEL
LIN {X 0,Y 441.729,Z 837.699,A -85,B 0,C 180,E1 -9167.83,E2 -9167.83} C_VEL
LIN {X 0,Y 441.222,Z 846.651,A -85,B 0,C 180,E1 -9168.981,E2 -9168.981} C_VEL
LIN {X 0,Y 440.807,Z 853.772,A -85,B 0,C 180,E1 -9170.131,E2 -9170.131} C_VEL
LIN {X 0,Y 440.444,Z 858.7,A -85,B 0,C 180,E1 -9171.05,E2 -9171.05} C_VEL
LIN {X 0,Y 440.167,Z 863.981,A -85,B 0,C 180,E1 -9172.229,E2 -9172.229} C_VEL
LIN {X 0,Y 439.838,Z 868.914,A -85,B 0,C 180,E1 -9173.578,E2 -9173.578} C_VEL
LIN {X 0,Y 439.52,Z 871.629,A -85,B 0,C 180,E1 -9174.495,E2 -9174.495} C_VEL
LIN {X 0,Y 439.349,Z 875.451,A -85,B 0,C 180,E1 -9176.331,E2 -9176.331} C_VEL
LIN {X 0,Y 439.342,Z 876.837,A -85,B 0,C 180,E1 -9177.249,E2 -9177.249} C_VEL
LIN {X 0,Y 439.125,Z 878.218,A -85,B 0,C 180,E1 -9179.083,E2 -9179.083} C_VEL
LIN {X 0,Y 439.106,Z 878.324,A -85,B 0,C 180,E1 -9180,E2 -9180} C_VEL
LIN {X 0,Y 439.082,Z 877.998,A -85,B 0,C 180,E1 -9180.917,E2 -9180.917} C_VEL
LIN {X 0,Y 439.067,Z 876.158,A -85,B 0,C 180,E1 -9182.752,E2 -9182.752} C_VEL
LIN {X 0,Y 439.276,Z 872.583,A -85,B 0,C 180,E1 -9184.588,E2 -9184.588} C_VEL
LIN {X 0,Y 439.462,Z 868.749,A -85,B 0,C 180,E1 -9185.967,E2 -9185.967} C_VEL
LIN {X 0,Y 439.738,Z 863.772,A -85,B 0,C 180,E1 -9187.346,E2 -9187.346} C_VEL
LIN {X 0,Y 439.991,Z 858.686,A -85,B 0,C 180,E1 -9188.497,E2 -9188.497} C_VEL
LIN {X 0,Y 440.387,Z 851.256,A -85,B 0,C 180,E1 -9189.878,E2 -9189.878} C_VEL
LIN {X 0,Y 440.693,Z 843.511,A -85,B 0,C 180,E1 -9191.033,E2 -9191.033} C_VEL
LIN {X 0,Y 441.074,Z 836.257,A -85,B 0,C 180,E1 -9191.955,E2 -9191.955} C_VEL
LIN {X 0,Y 441.391,Z 828.877,A -85,B 0,C 180,E1 -9192.763,E2 -9192.763} C_VEL
LIN {X 0,Y 441.893,Z 818.857,A -85,B 0,C 180,E1 -9193.685,E2 -9193.685} C_VEL
LIN {X 0,Y 442.242,Z 809.649,A -85,B 0,C 180,E1 -9194.366,E2 -9194.366} C_VEL
LIN {X 0,Y 441.663,Z 806.055,A -85,B 0,C 180,E1 -9194.628,E2 -9194.628} C_VEL
LIN {X 0,Y 439.412,Z 797.752,A -85,B 0,C 180,E1 -9195.213,E2 -9195.213} C_VEL
LIN {X 0,Y 439.372,Z 797.75,A -85,B 0,C 180,E1 -9198.658,E2 -9198.658} C_VEL
LIN {X 0,Y 439.384,Z 797.751,A -85,B 0,C 180,E1 -9201.916,E2 -9201.916} C_VEL
LIN {X 0,Y 439.38,Z 797.749,A -85,B 0,C 180,E1 -9204.575,E2 -9204.575} C_VEL
LIN {X 0,Y 439.337,Z 797.755,A -85,B 0,C 180,E1 -9207.64,E2 -9207.64} C_VEL
LIN {X 0,Y 439.36,Z 797.75,A -85,B 0,C 180,E1 -9210.789,E2 -9210.789} C_VEL
LIN {X 0,Y 439.382,Z 797.754,A -85,B 0,C 180,E1 -9214.044,E2 -9214.044} C_VEL
LIN {X 0,Y 439.343,Z 797.751,A -85,B 0,C 180,E1 -9216.884,E2 -9216.884} C_VEL
LIN {X 0,Y 439.351,Z 797.758,A -85,B 0,C 180,E1 -9219.84,E2 -9219.84} C_VEL
LIN {X 0,Y 439.341,Z 797.754,A -85,B 0,C 180,E1 -9222.62,E2 -9222.62} C_VEL
LIN {X 0,Y 439.405,Z 797.747,A -85,B 0,C 180,E1 -9225.27,E2 -9225.27} C_VEL
LIN {X 0,Y 439.377,Z 797.751,A -85,B 0,C 180,E1 -9228.745,E2 -9228.745} C_VEL
LIN {X 0,Y 439.37,Z 797.753,A -85,B 0,C 180,E1 -9231.609,E2 -9231.609} C_VEL
LIN {X 0,Y 439.402,Z 797.748,A -85,B 0,C 180,E1 -9234.843,E2 -9234.843} C_VEL
LIN {X 0,Y 439.378,Z 797.755,A -85,B 0,C 180,E1 -9238.139,E2 -9238.139} C_VEL
LIN {X 0,Y 439.439,Z 797.74,A -85,B 0,C 180,E1 -9241.597,E2 -9241.597} C_VEL
LIN {X 0,Y 439.393,Z 797.75,A -85,B 0,C 180,E1 -9244.413,E2 -9244.413} C_VEL
LIN {X 0,Y 439.37,Z 797.752,A -85,B 0,C 180,E1 -9247.423,E2 -9247.423} C_VEL
LIN {X 0,Y 439.447,Z 797.751,A -85,B 0,C 180,E1 -9250.662,E2 -9250.662} C_VEL
LIN {X 0,Y 439.487,Z 797.741,A -85,B 0,C 180,E1 -9254.343,E2 -9254.343} C_VEL
LIN {X 0,Y 439.526,Z 798.075,A -85,B 0,C 180,E1 -9254.404,E2 -9254.404} C_VEL
LIN {X 0,Y 442.882,Z 809.336,A -85,B 0,C 180,E1 -9255.173,E2 -9255.173} C_VEL
LIN {X 0,Y 443.161,Z 812.387,A -85,B 0,C 180,E1 -9255.39,E2 -9255.39} C_VEL
LIN {X 0,Y 442.672,Z 823.456,A -85,B 0,C 180,E1 -9256.221,E2 -9256.221} C_VEL
LIN {X 0,Y 442.196,Z 833.242,A -85,B 0,C 180,E1 -9257.142,E2 -9257.142} C_VEL
LIN {X 0,Y 441.643,Z 843.087,A -85,B 0,C 180,E1 -9258.292,E2 -9258.292} C_VEL
LIN {X 0,Y 440.996,Z 852.588,A -85,B 0,C 180,E1 -9259.67,E2 -9259.67} C_VEL
LIN {X 0,Y 440.503,Z 860.155,A -85,B 0,C 180,E1 -9261.05,E2 -9261.05} C_VEL
LIN {X 0,Y 440.332,Z 863.491,A -85,B 0,C 180,E1 -9261.776,E2 -9261.776} C_VEL
LIN {X 0,Y 439.454,Z 866.39,A -85,B 0,C 180,E1 -9262.44,E2 -9262.44} C_VEL
LIN {X 0,Y 436.349,Z 870.857,A -85,B 0,C 180,E1 -9263.526,E2 -9263.526} C_VEL
LIN {X 0,Y 433.281,Z 874.623,A -85,B 0,C 180,E1 -9264.664,E2 -9264.664} C_VEL
LIN {X 0,Y 432.476,Z 876.365,A -85,B 0,C 180,E1 -9265.403,E2 -9265.403} C_VEL
LIN {X 0,Y 432.348,Z 878.059,A -85,B 0,C 180,E1 -9266.27,E2 -9266.27} C_VEL
LIN {X 0,Y 432.355,Z 879.416,A -85,B 0,C 180,E1 -9267.203,E2 -9267.203} C_VEL
LIN {X 0,Y 432.264,Z 880.99,A -85,B 0,C 180,E1 -9269.067,E2 -9269.067} C_VEL
LIN {X 0,Y 432.263,Z 881.219,A -85,B 0,C 180,E1 -9269.998,E2 -9269.998} C_VEL
LIN {X 0,Y 432.256,Z 881.04,A -85,B 0,C 180,E1 -9270.93,E2 -9270.93} C_VEL
LIN {X 0,Y 432.352,Z 879.532,A -85,B 0,C 180,E1 -9272.793,E2 -9272.793} C_VEL
LIN {X 0,Y 432.341,Z 878.226,A -85,B 0,C 180,E1 -9273.726,E2 -9273.726} C_VEL
LIN {X 0,Y 432.552,Z 875.424,A -85,B 0,C 180,E1 -9275.125,E2 -9275.125} C_VEL
LIN {X 0,Y 432.983,Z 871.599,A -85,B 0,C 180,E1 -9276.522,E2 -9276.522} C_VEL
LIN {X 0,Y 433.299,Z 866.362,A -85,B 0,C 180,E1 -9278.01,E2 -9278.01} C_VEL
LIN {X 0,Y 433.683,Z 859.332,A -85,B 0,C 180,E1 -9279.56,E2 -9279.56} C_VEL
LIN {X 0,Y 434.294,Z 851.314,A -85,B 0,C 180,E1 -9280.959,E2 -9280.959} C_VEL
LIN {X 0,Y 434.847,Z 843.095,A -85,B 0,C 180,E1 -9282.127,E2 -9282.127} C_VEL
LIN {X 0,Y 435.384,Z 832.933,A -85,B 0,C 180,E1 -9283.297,E2 -9283.297} C_VEL
LIN {X 0,Y 436.106,Z 821.951,A -85,B 0,C 180,E1 -9284.299,E2 -9284.299} C_VEL
LIN {X 0,Y 436.281,Z 811.799,A -85,B 0,C 180,E1 -9285.054,E2 -9285.054} C_VEL
LIN {X 0,Y 433.007,Z 800.662,A -85,B 0,C 180,E1 -9285.856,E2 -9285.856} C_VEL
LIN {X 0,Y 432.421,Z 798.623,A -85,B 0,C 180,E1 -9286.007,E2 -9286.007} C_VEL
LIN {X 0,Y 432.385,Z 798.625,A -85,B 0,C 180,E1 -9289.483,E2 -9289.483} C_VEL
LIN {X 0,Y 432.317,Z 798.63,A -85,B 0,C 180,E1 -9292.962,E2 -9292.962} C_VEL
LIN {X 0,Y 432.361,Z 798.631,A -85,B 0,C 180,E1 -9296.03,E2 -9296.03} C_VEL
LIN {X 0,Y 432.339,Z 798.628,A -85,B 0,C 180,E1 -9299.185,E2 -9299.185} C_VEL
LIN {X 0,Y 432.317,Z 798.634,A -85,B 0,C 180,E1 -9302.441,E2 -9302.441} C_VEL
LIN {X 0,Y 432.338,Z 798.63,A -85,B 0,C 180,E1 -9305.63,E2 -9305.63} C_VEL
LIN {X 0,Y 432.35,Z 798.628,A -85,B 0,C 180,E1 -9308.715,E2 -9308.715} C_VEL
LIN {X 0,Y 432.365,Z 798.626,A -85,B 0,C 180,E1 -9311.79,E2 -9311.79} C_VEL
LIN {X 0,Y 432.368,Z 798.63,A -85,B 0,C 180,E1 -9314.34,E2 -9314.34} C_VEL
LIN {X 0,Y 432.355,Z 798.623,A -85,B 0,C 180,E1 -9317.007,E2 -9317.007} C_VEL
LIN {X 0,Y 432.347,Z 798.627,A -85,B 0,C 180,E1 -9319.815,E2 -9319.815} C_VEL
LIN {X 0,Y 432.305,Z 798.633,A -85,B 0,C 180,E1 -9323.022,E2 -9323.022} C_VEL
LIN {X 0,Y 432.346,Z 798.623,A -85,B 0,C 180,E1 -9325.995,E2 -9325.995} C_VEL
LIN {X 0,Y 432.381,Z 798.618,A -85,B 0,C 180,E1 -9329.743,E2 -9329.743} C_VEL
LIN {X 0,Y 432.385,Z 798.621,A -85,B 0,C 180,E1 -9333.371,E2 -9333.371} C_VEL
LIN {X 0,Y 432.356,Z 798.624,A -85,B 0,C 180,E1 -9336.022,E2 -9336.022} C_VEL
LIN {X 0,Y 432.334,Z 798.631,A -85,B 0,C 180,E1 -9339.045,E2 -9339.045} C_VEL
LIN {X 0,Y 432.361,Z 798.624,A -85,B 0,C 180,E1 -9342.01,E2 -9342.01} C_VEL
LIN {X 0,Y 432.378,Z 798.622,A -85,B 0,C 180,E1 -9344.926,E2 -9344.926} C_VEL
LIN {X 0,Y 432.465,Z 798.613,A -85,B 0,C 180,E1 -9347.804,E2 -9347.804} C_VEL
LIN {X 0,Y 432.475,Z 798.614,A -85,B 0,C 180,E1 -9351.59,E2 -9351.59} C_VEL
LIN {X 0,Y 432.576,Z 798.6,A -85,B 0,C 180,E1 -9354.406,E2 -9354.406} C_VEL
LIN {X 0,Y 432.587,Z 798.598,A -85,B 0,C 180,E1 -9358.138,E2 -9358.138} C_VEL
LIN {X 0,Y 432.714,Z 798.584,A -85,B 0,C 180,E1 -9360,E2 -9360} C_VEL
LIN {X 0,Y 432.575,Z 798.6,A -85,B 0,C 180,E1 -9362.794,E2 -9362.794} C_VEL
LIN {X 0,Y 432.566,Z 798.607,A -85,B 0,C 180,E1 -9365.594,E2 -9365.594} C_VEL
LIN {X 0,Y 432.465,Z 798.612,A -85,B 0,C 180,E1 -9368.41,E2 -9368.41} C_VEL
LIN {X 0,Y 432.463,Z 798.611,A -85,B 0,C 180,E1 -9372.196,E2 -9372.196} C_VEL
LIN {X 0,Y 432.412,Z 798.625,A -85,B 0,C 180,E1 -9376.04,E2 -9376.04} C_VEL
LIN {X 0,Y 432.369,Z 798.627,A -85,B 0,C 180,E1 -9379.486,E2 -9379.486} C_VEL
LIN {X 0,Y 432.3,Z 798.633,A -85,B 0,C 180,E1 -9382.965,E2 -9382.965} C_VEL
LIN {X 0,Y 432.32,Z 798.629,A -85,B 0,C 180,E1 -9385.003,E2 -9385.003} C_VEL
LIN {X 0,Y 432.327,Z 798.633,A -85,B 0,C 180,E1 -9388.127,E2 -9388.127} C_VEL
LIN {X 0,Y 432.305,Z 798.632,A -85,B 0,C 180,E1 -9391.347,E2 -9391.347} C_VEL
LIN {X 0,Y 432.312,Z 798.635,A -85,B 0,C 180,E1 -9394.68,E2 -9394.68} C_VEL
LIN {X 0,Y 432.308,Z 798.637,A -85,B 0,C 180,E1 -9398.153,E2 -9398.153} C_VEL
LIN {X 0,Y 432.292,Z 798.635,A -85,B 0,C 180,E1 -9401.802,E2 -9401.802} C_VEL
LIN {X 0,Y 432.319,Z 798.632,A -85,B 0,C 180,E1 -9404.349,E2 -9404.349} C_VEL
LIN {X 0,Y 432.311,Z 798.784,A -85,B 0,C 180,E1 -9407.717,E2 -9407.717} C_VEL
LIN {X 0,Y 434.166,Z 807.824,A -85,B 0,C 180,E1 -9410.567,E2 -9410.567} C_VEL
LIN {X 0,Y 435.625,Z 815.487,A -85,B 0,C 180,E1 -9412.845,E2 -9412.845} C_VEL
LIN {X 0,Y 435.524,Z 821.479,A -85,B 0,C 180,E1 -9414.487,E2 -9414.487} C_VEL
LIN {X 0,Y 434.798,Z 833.971,A -85,B 0,C 180,E1 -9417.767,E2 -9417.767} C_VEL
LIN {X 0,Y 433.991,Z 849.597,A -85,B 0,C 180,E1 -9421.732,E2 -9421.732} C_VEL
LIN {X 0,Y 433.445,Z 861.968,A -85,B 0,C 180,E1 -9424.812,E2 -9424.812} C_VEL
LIN {X 0,Y 432.848,Z 875.191,A -85,B 0,C 180,E1 -9428.074,E2 -9428.074} C_VEL
LIN {X 0,Y 432.411,Z 889.16,A -85,B 0,C 180,E1 -9431.524,E2 -9431.524} C_VEL
LIN {X 0,Y 432.147,Z 896.103,A -85,B 0,C 180,E1 -9433.253,E2 -9433.253} C_VEL
LIN {X 0,Y 433.684,Z 911.337,A -85,B 0,C 180,E1 -9433.725,E2 -9433.725} C_VEL
LIN {X 0,Y 434.773,Z 922.741,A -85,B 0,C 180,E1 -9434.232,E2 -9434.232} C_VEL
LIN {X 0,Y 435.117,Z 927.466,A -85,B 0,C 180,E1 -9434.485,E2 -9434.485} C_VEL
LIN {X 0,Y 434.476,Z 939.877,A -85,B 0,C 180,E1 -9435.242,E2 -9435.242} C_VEL
LIN {X 0,Y 433.789,Z 951.477,A -85,B 0,C 180,E1 -9436.163,E2 -9436.163} C_VEL
LIN {X 0,Y 433.264,Z 962.24,A -85,B 0,C 180,E1 -9437.233,E2 -9437.233} C_VEL
LIN {X 0,Y 432.674,Z 970.928,A -85,B 0,C 180,E1 -9438.287,E2 -9438.287} C_VEL
LIN {X 0,Y 432.218,Z 978.975,A -85,B 0,C 180,E1 -9439.461,E2 -9439.461} C_VEL
LIN {X 0,Y 431.875,Z 986.87,A -85,B 0,C 180,E1 -9440.872,E2 -9440.872} C_VEL
LIN {X 0,Y 431.729,Z 992.297,A -85,B 0,C 180,E1 -9442.048,E2 -9442.048} C_VEL
